Omron Sysmac Studio project Auto Connect Project (Sysmac Studio 1.61.0.64007, StandardProject)

# Controller new_Controller_0: NX102-9000 version 1.68
Units and slaves: 유니트 1 : NX-PF0730 (N1); 유니트 2 : NX-CIF105 (N2); 유니트 3 : NX-ID5342 (N3); 유니트 4 : NX-OD5121 (N4); 유니트 5 : NX-OD5121 (N5)
Task PrimaryTask (priority 4, period or condition 1000): Program0
Library MTCP_Server_NJNX 2.6. (contents left out)

TYPE sStepControl : STRUCT
    MoveStart : BOOL;
    TargetPulse : INT;  (* Unit : pulse *)
    SetDir : BOOL;  (* TRUE : CW, FALSE, CCW *)
END_STRUCT END_TYPE
TYPE sMotor : STRUCT
    Up : BOOL;
    Down : BOOL;
    Origin : BOOL;
    Move : INT;  (* Unit: 0.1 mm *)
    Check : BOOL;  (* Checking variable whether TRUE of FALSE *)
    Seq : INT;  (* Sequence Index *)
END_STRUCT END_TYPE
TYPE sModule : STRUCT
    Input : sModuleInput;
    Output : sModuleOutput;
END_STRUCT END_TYPE
TYPE sModuleInput : STRUCT
    Command : sModuleInputCommand;
END_STRUCT END_TYPE
TYPE sModuleOutput : STRUCT
    Status : sModuleOutputStatus;
END_STRUCT END_TYPE
TYPE sModuleInputCommand : STRUCT
    bCylinder1Down : BOOL;
    bCylinder1Up : BOOL;
END_STRUCT END_TYPE
TYPE sModuleOutputStatus : STRUCT
    bCylinder1Down : BOOL;
    bCylinder1Up : BOOL;
END_STRUCT END_TYPE

TYPE typeOPC\sProdTracker : STRUCT
    Input : typeOPC\sProdTrackerInput;
    Output : typeOPC\sProdTrackerOutput;
    Capture : typeOPC\sProdTrackerCapture;
    PTZ : typeOPC\sProdTrackerPTZ;
END_STRUCT END_TYPE
TYPE typeOPC\sProdTrackerInput : STRUCT
    nStart : INT;
    strData : STRING[256];
    nResult : INT;
END_STRUCT END_TYPE
TYPE typeOPC\sProdTrackerOutput : STRUCT
    nResponse : INT;
    dtUpdateTime : DATE_AND_TIME;
END_STRUCT END_TYPE
TYPE typeOPC\sProdTrackerCapture : STRUCT
    bStart : BOOL;
    strData : STRING[256];
END_STRUCT END_TYPE
TYPE typeOPC\sProdTrackerPTZ : STRUCT
    bStart : BOOL;
    nPreset : INT;
END_STRUCT END_TYPE

TYPE Data\sOT2 : STRUCT
    Pipette0 : INT;  (* 총 96개 pipette *)
    Pipette1 : INT;  (* 총 96개 pipette *)
    BigVial0 : Data\sBigVial;  (* 총 6개 바이알 *)
    BigVial1 : Data\sBigVial;  (* 총 6개 바이알 *)
    WellPlate : INT;  (* 총 96개 well *)
    HeatPlate : Data\sHeatPlate;  (* 총 12개 well *)
    OT2Job : STRING[256];  (* OT2 현황 *)
END_STRUCT END_TYPE
TYPE Data\sBigVial : STRUCT
    BVname : ARRAY[0..5] OF STRING[256];
    BVvolume : ARRAY[0..5] OF REAL;
END_STRUCT END_TYPE
TYPE Data\sHeatPlate : STRUCT
    HPname : ARRAY[0..11] OF STRING[256];
    HPvolume : ARRAY[0..11] OF REAL;
END_STRUCT END_TYPE
TYPE Data\sCell : STRUCT
    CSASstack : INT;  (* 양극, 스프링, 음극, 분리막 스태킹 구조물 (총 4개) *)
    CCSstack : INT;  (* 캔, 캡, 스페이서 스태킹 구조물 (총 4개) *)
    CScomp : INT;  (* 양극, 스프링 회전 구조물 (총 12개) *)
    AScomp : INT;  (* 음극, 분리막 회전 구조물 (총 12개) *)
    CCScomp : INT;  (* 캔, 캡, 스페이서 액츄에이터 구조물 (총 12개) *)
    Assembly : STRING[256];  (* 셀 조립대의 현황 (ex. can or sep or liquid) *)
    Crimper : BOOL;  (* 크림퍼 내 셀 존재 유무 *)
END_STRUCT END_TYPE
TYPE Data\sJig : STRUCT
    Cycler : Data\sCycler;
    EIS : Data\sEIS;
    Gantry : ARRAY[0..1] OF STRING[256];  (* 현재 직교로봇이 진행중인 작업 (ex. [EIS_Insert, 0]) *)
END_STRUCT END_TYPE
TYPE Data\sCycler : STRUCT
    name : ARRAY[0..47] OF STRING[256];  (* Cycling 셀 이름 *)
    status : ARRAY[0..47] OF STRING[256];  (* Cycler 현황 (empty, in, cycling, done) *)
END_STRUCT END_TYPE
TYPE Data\sEIS : STRUCT
    name : ARRAY[0..1] OF STRING[256];  (* EIS 셀 이름 *)
    status : ARRAY[0..1] OF STRING[256];  (* EIS 현황 (empty, in, cycling, done) *)
END_STRUCT END_TYPE

VAR_GLOBAL CONSTANT
    N1_Node_location_information : _sNXUNIT_ID := (NodeAdr := 65535, IPAdr := [5(16#FF)], UnitNo := 2, Path := [16#1, 16#0, 16#2, 16#0, 16#2, 59(16#0)], PathLength := 6);
END_VAR
VAR_GLOBAL
    Pulse0 : BOOL;  (* at IOBus://unit#5/Output Bit 16 bits/Output Bit 01 *)
    Direction0 : BOOL;  (* at IOBus://unit#5/Output Bit 16 bits/Output Bit 00 *)
    Pulse1 : BOOL;  (* at IOBus://unit#5/Output Bit 16 bits/Output Bit 03 *)
    Direction1 : BOOL;  (* at IOBus://unit#5/Output Bit 16 bits/Output Bit 02 *)
    Pulse2 : BOOL;  (* at IOBus://unit#5/Output Bit 16 bits/Output Bit 05 *)
    Direction2 : BOOL;  (* at IOBus://unit#5/Output Bit 16 bits/Output Bit 04 *)
    Pulse3 : BOOL;  (* at IOBus://unit#5/Output Bit 16 bits/Output Bit 07 *)
    Direction3 : BOOL;  (* at IOBus://unit#5/Output Bit 16 bits/Output Bit 06 *)
    Pulse4 : BOOL;  (* Front Z; at IOBus://unit#5/Output Bit 16 bits/Output Bit 09 *)
    Direction4 : BOOL;  (* Front Z; at IOBus://unit#5/Output Bit 16 bits/Output Bit 08 *)
    Pulse5 : BOOL;  (* Front X; at IOBus://unit#5/Output Bit 16 bits/Output Bit 11 *)
    Direction5 : BOOL;  (* Front X; at IOBus://unit#5/Output Bit 16 bits/Output Bit 10 *)
    Pulse6 : BOOL;  (* Back Z; at IOBus://unit#5/Output Bit 16 bits/Output Bit 13 *)
    Direction6 : BOOL;  (* Back Z; at IOBus://unit#5/Output Bit 16 bits/Output Bit 12 *)
    Pulse7 : BOOL;  (* Back X; at IOBus://unit#5/Output Bit 16 bits/Output Bit 15 *)
    Direction7 : BOOL;  (* Back X; at IOBus://unit#5/Output Bit 16 bits/Output Bit 14 *)
    Sensor0 : BOOL;  (* Rotary for Cathode&Spring; at IOBus://unit#3/Input Bit 16 bits/Input Bit 12 *)
    Sensor1 : BOOL;  (* Rotary for Anode&Separator; at IOBus://unit#3/Input Bit 16 bits/Input Bit 13 *)
    Sensor2 : BOOL;  (* Stacking for CSAS; at IOBus://unit#3/Input Bit 16 bits/Input Bit 14 *)
    Sensor3 : BOOL;  (* Stacking for Can&Cap&Spacer; at IOBus://unit#3/Input Bit 16 bits/Input Bit 15 *)
    Sensor4_L : BOOL;  (* Front Z; at IOBus://unit#3/Input Bit 16 bits/Input Bit 01 *)
    Sensor4_R : BOOL;  (* Front Z; at IOBus://unit#3/Input Bit 16 bits/Input Bit 02 *)
    Sensor5_L : BOOL;  (* Front X; at IOBus://unit#3/Input Bit 16 bits/Input Bit 04 *)
    Sensor5_R : BOOL;  (* Front X; at IOBus://unit#3/Input Bit 16 bits/Input Bit 05 *)
    Sensor6_L : BOOL;  (* Back Z; at IOBus://unit#3/Input Bit 16 bits/Input Bit 07 *)
    Sensor6_R : BOOL;  (* Back Z; at IOBus://unit#3/Input Bit 16 bits/Input Bit 08 *)
    Sensor7_L : BOOL;  (* Back X; at IOBus://unit#3/Input Bit 16 bits/Input Bit 10 *)
    Sensor7_R : BOOL;  (* Back X; at IOBus://unit#3/Input Bit 16 bits/Input Bit 11 *)
    ENA0 : BOOL;  (* at IOBus://unit#4/Output Bit 16 bits/Output Bit 01 *)
    ENA1 : BOOL;  (* at IOBus://unit#4/Output Bit 16 bits/Output Bit 03 *)
    ENA2 : BOOL;  (* at IOBus://unit#4/Output Bit 16 bits/Output Bit 05 *)
    ENA3 : BOOL;  (* at IOBus://unit#4/Output Bit 16 bits/Output Bit 07 *)
    ENA4 : BOOL;  (* at IOBus://unit#4/Output Bit 16 bits/Output Bit 09 *)
    ENA5 : BOOL;  (* at IOBus://unit#4/Output Bit 16 bits/Output Bit 11 *)
    ENA6 : BOOL;  (* at IOBus://unit#4/Output Bit 16 bits/Output Bit 13 *)
    ENA7 : BOOL;  (* at IOBus://unit#4/Output Bit 16 bits/Output Bit 15 *)
    RELAY0 : BOOL;  (* For STEP Motor; at IOBus://unit#4/Output Bit 16 bits/Output Bit 00 *)
    RELAY1 : BOOL;  (* For Crimper; at IOBus://unit#4/Output Bit 16 bits/Output Bit 02 *)
    Sensor4_O : BOOL;  (* Front Z *)
    Sensor5_O : BOOL;  (* Front X; at IOBus://unit#3/Input Bit 16 bits/Input Bit 03 *)
    Sensor6_O : BOOL;  (* Back Z; at IOBus://unit#3/Input Bit 16 bits/Input Bit 06 *)
    Sensor7_O : BOOL;  (* Back X; at IOBus://unit#3/Input Bit 16 bits/Input Bit 09 *)
    Robot_moving : BOOL;  (* True: Robot moving, False: Robot stop; at IOBus://unit#3/Input Bit 16 bits/Input Bit 00; published *)
    Motor0_Up : BOOL;  (* published *)
    Motor0_Down : BOOL;  (* published *)
    Motor0_Origin : BOOL;  (* published *)
    Motor0_Move : INT;  (* published *)
END_VAR
VAR_GLOBAL RETAIN
    Motor0_Check : BOOL;  (* published *)
END_VAR
VAR_GLOBAL
    Motor1_Up : BOOL;  (* published *)
    Motor1_Down : BOOL;  (* published *)
    Motor1_Origin : BOOL;  (* published *)
    Motor1_Move : INT;  (* published *)
    Motor1_Check : BOOL;  (* published *)
    Motor2_Up : BOOL;  (* published *)
    Motor2_Down : BOOL;  (* published *)
    Motor2_Origin : BOOL;  (* published *)
    Motor2_Move : INT;  (* published *)
    Motor2_Check : BOOL;  (* published *)
    Motor3_Up : BOOL;  (* published *)
    Motor3_Down : BOOL;  (* published *)
    Motor3_Origin : BOOL;  (* published *)
    Motor3_Move : INT;  (* published *)
    Motor3_Check : BOOL;  (* published *)
    Motor4_Up : BOOL;  (* published *)
    Motor4_Down : BOOL;  (* published *)
    Motor4_Origin : BOOL;  (* published *)
    Motor4_Move : INT;  (* 1 = 0.1 mm (ex. 25 = 2.5 mm); published *)
    Motor4_Check : BOOL;  (* published *)
    Motor5_Up : BOOL;  (* published *)
    Motor5_Down : BOOL;  (* published *)
    Motor5_Origin : BOOL;  (* published *)
    Motor5_Move : INT;  (* 1 = 0.1 mm (ex. 25 = 2.5 mm); published *)
    Motor5_Check : BOOL;  (* published *)
    Motor6_Up : BOOL;  (* published *)
    Motor6_Down : BOOL;  (* published *)
    Motor6_Origin : BOOL;  (* published *)
    Motor6_Move : INT;  (* 1 = 0.1 mm (ex. 25 = 2.5 mm); published *)
    Motor6_Check : BOOL;  (* published *)
    Motor7_Up : BOOL;  (* published *)
    Motor7_Down : BOOL;  (* published *)
    Motor7_Origin : BOOL;  (* published *)
    Motor7_Move : INT;  (* 1 = 0.1 mm (ex. 25 = 2.5 mm); published *)
    Motor7_Check : BOOL;  (* published *)
    Jigmove_csv : ARRAY[0..47,0..5] OF REAL;  (* for coincell Jig; published *)
    EISmove_csv : ARRAY[0..1,0..3] OF REAL;  (* for EIS Jig; published *)
    JigIndex : INT;  (* Jig: 0~47; published *)
    EISIndex : INT;  (* EIS: 0~1; published *)
    ActuIndex : INT;  (* published *)
    ActuMove : INT;  (* published *)
    Open_Serial : BOOL;  (* published *)
    PS2_Data : ARRAY[0..19] OF WORD;  (* Modbus TCP Write Data; published *)
    Open_MB : BOOL;  (* Modbus TCP Write; published *)
    Crimper_Done : BOOL;  (* published *)
    Crimper_On : BOOL;  (* published *)
    Jig_Readypos : BOOL;  (* published *)
    Jig_Insert : BOOL;  (* published *)
    Jig_Retrieve : BOOL;  (* published *)
    Robot_moving2 : BOOL;  (* 직접 지정 가능한 Robot moving Bool; published *)
    CCSactu_Check : BOOL;  (* 캔, 캡, 스페이서 액츄에이터 동작; published *)
    CCSactu_Index : INT;  (* 0: 원점, 1~12: 해당 위치만큼 올림; published *)
    CCSalign_Check : BOOL;  (* 캔, 캡, 스페이서 정렬 동작; published *)
    Assemalign_Check : BOOL;  (* 셀 조립대 정렬 동작; published *)
    JOBList : ARRAY[0..299] OF STRING[256];  (* 던져진 JOB 을 정리한 리스트; published *)
    JOB : ARRAY[0..1] OF STRING[256];  (* 지그에 던지는 JOB; published *)
    JOB_Done : BOOL;  (* True 면 지그에 던져진 다음 작업 수행; published *)
    Readypos_Done : BOOL;  (* 지그가 셀 받을 대기 상태; published *)
    Coincell_Job : ARRAY[0..47,0..9] OF BOOL;  (* 1열 셀 삽입(True: 셀 삽입됨), 2열: 1번 조건 완료, 3열: 2번 조건 완료...; published *)
    Coincell_EISJob : ARRAY[0..1,0..1] OF BOOL;  (* 1열 셀 삽입(True: 셀 삽입됨), 2열: 셀 평가 완료(True: 셀 평가 완료됨); published *)
    Coincell_Return : ARRAY[0..1] OF INT;  (* EIS 측정 후 돌아가야 할 포지션 위치; published *)
    ProdTracker : typeOPC\sProdTracker;  (* 카메라 (ProdTracker); published *)
    DataOT2 : Data\sOT2;  (* OT2 관련 데이터; published *)
    DataCell : Data\sCell;  (* 셀 조립 관련 데이터; published *)
    DataJig : Data\sJig;  (* 셀 지그 관련 데이터; published *)
END_VAR

PROGRAM Program0
VAR
    Open_Port : BOOL;
    Port_Open : BOOL;
    Port_Busy : BOOL;
    Port_Error : BOOL;
    Port_ErrorID : WORD;
    MB_Socket : _sSOCKET;
    do_nothing : BOOL;
    MBTCP_FN3 : ModbusTCPRead;
    Open_Socket : SktTCPConnect;
    FN3_Read_Cmd : _sMODBUS_READ;
    PS_Data : ARRAY[0..15] OF WORD;
    FN3_Busy : BOOL;
    FN3_Error : BOOL;
    FN3_ErrorID : WORD;
    FN3_Erridx : DWORD;
    Read_Size : UINT;
    do_nothing2 : BOOL;
    MBTCP_FN4 : ModbusTCPWrite;
    FN4_Write_Cmd : _sMODBUS_WRITE;
    FN4_Busy : BOOL;
    FN4_Error : BOOL;
    FN4_ErrorID : WORD;
    FN4_Erridx : DWORD;
    Open_RTU : BOOL;
    MBRTU_FN3 : NX_ModbusRtuWrite;
    MBRTU_FN1 : NX_ModbusRtuWrite;
    MBRTU_FN5 : NX_ModbusRtuWrite;
    FN5_Write_Cmd : _sSERIAL_MODBUSRTU_WRITE;
    PS5_Data : WORD;
    FN5_Port : _sDEVICE_PORT;
    FN5_Busy : BOOL;
    FN5_CmdAbort : BOOL;
    FN5_Error : BOOL;
    FN5_ErrorID : WORD;
    FN5_Erridx : DWORD;
    do_nothing3 : BOOL;
    RTUSlaveAdr : UINT := 11;
    bOutputStart : BOOL;
    bOutput : BOOL;
    nCount : INT;
    maxCount : INT;
    Open_Server : BOOL;
    TCPServer : MTCP_Server_NJNX;
    Server_Connected : BOOL;
    Reset_SdRcvCnt : BOOL := False;
    SdRcv_Cnt : UDINT;
    Port_Client : UINT;
    IP_Client : STRING[24];
    TCP_Status : _eCONNECTION_STATE;
    ErrorID : WORD;
    Error : BOOL;
    MotorStart : BOOL;
    TON_test : TON;
    TP_test : TP;
    FB_Motor1_Control : STEPmotor;
    Delay_TON0 : TON;
    o : BOOL;
    Motor1Control : sStepControl;
    FB_Motor0_Control : STEPmotor;
    Motor0Control : sStepControl;
    FB_Motor2_Control : STEPmotor;
    Motor2Control : sStepControl;
    Motor4Control : sStepControl;
    MotorRelay : BOOL;
    FB_Motor4_Control : STEPmotor;
    FB_Motor5_Control : STEPmotor;
    Motor5Control : sStepControl;
    FB_Motor6_Control : STEPmotor;
    Motor6Control : sStepControl;
    FB_Motor7_Control : STEPmotor;
    Motor7Control : sStepControl;
    Motor0 : sMotor;
    Motor1 : sMotor;
    Motor2 : sMotor;
    Motor3 : sMotor;
    Motor4 : sMotor;
    Motor5 : sMotor;
    Motor6 : sMotor;
    Motor7 : sMotor;
    FB_Motor3_Control : STEPmotor;
    Motor3Control : sStepControl;
    Open_MBRead : BOOL;
    bDebugBit : BOOL;
    Serial_FN6 : NX_SerialSend;
    do_nothing4 : BOOL;
    FN6_Port : _sDEVICE_PORT;
    Serial_Error : BOOL;
    Serial_Errid : WORD;
    Serial_Busy : BOOL;
    SendSize : UINT := 10;
    Jig_Origin : BOOL;
    Jig_Seq : INT;
    SendData : ARRAY[0..9] OF BYTE;
    JigOrigin_Seq : INT;
    chksum : BYTE;
    test : BOOL;
    Test_Seq : INT;
    JigReady_Seq : INT;
    Finish0 : BOOL;
    Finish1 : BOOL;
    Finish2 : BOOL;
    Finish3 : BOOL;
    Finish4 : BOOL;
    Finish5 : BOOL;
    Finish6 : BOOL;
    Finish7 : BOOL;
    JigRetrieve_Seq : INT;
    Crimper_Seq : INT;
    EIS_Seq : INT;
    EIS_Insert : BOOL;
    EISRetrieve_Seq : INT;
    EIS_Retrieve : BOOL;
    Delay_TON1 : TON;
    Delay_TON6 : TON;
    Delay_TON7 : TON;
    Delay_TON8 : TON;
    Delay_TON9 : TON;
    Delay_TON10 : TON;
    Delay_TON11 : TON;
    Delay_TON12 : TON;
    Delay_TON13 : TON;
    Delay_TON2 : TON;
    Delay_TON3 : TON;
    Delay_TON4 : TON;
    Delay_TON5 : TON;
    Delay_TON14 : TON;
    CCSactu_seq : INT;
    Delay_TON15 : TON;
    CCSalign_seq : INT;
    Delay_TON16 : TON;
    Assemalign_seq : INT;
    Delay_TON17 : TON;
    JOB_seq : INT;
    i : INT;
    JOBList_Clear : BOOL;
    JOBprocesstest : BOOL;
    JOBDone_Check : BOOL;
    SendData4 : BYTE := 05;
    SendData5 : BYTE := 243;
    SendData6 : BYTE := 134;
END_VAR
VAR_EXTERNAL CONSTANT
    N1_Node_location_information : _sNXUNIT_ID;
END_VAR
VAR_EXTERNAL
    Pulse0 : BOOL;
    Direction0 : BOOL;
    Pulse1 : BOOL;
    Direction1 : BOOL;
    ENA0 : BOOL;
    ENA1 : BOOL;
    ENA2 : BOOL;
    ENA3 : BOOL;
    ENA4 : BOOL;
    ENA5 : BOOL;
    ENA6 : BOOL;
    ENA7 : BOOL;
    RELAY0 : BOOL;
    Direction2 : BOOL;
    Direction3 : BOOL;
    Pulse2 : BOOL;
    Pulse3 : BOOL;
    Sensor0 : BOOL;
    Sensor1 : BOOL;
    Direction5 : BOOL;
    Pulse5 : BOOL;
    Sensor3 : BOOL;
    Sensor2 : BOOL;
    Direction4 : BOOL;
    Pulse4 : BOOL;
    Direction6 : BOOL;
    Pulse6 : BOOL;
    Direction7 : BOOL;
    Pulse7 : BOOL;
    Sensor4_L : BOOL;
    Sensor6_L : BOOL;
    Sensor4_R : BOOL;
    Sensor6_R : BOOL;
    Sensor5_L : BOOL;
    Sensor5_R : BOOL;
    Sensor7_L : BOOL;
    Sensor7_R : BOOL;
    Robot_moving : BOOL;
    Motor0_Up : BOOL;
    Motor0_Down : BOOL;
    Motor0_Origin : BOOL;
    Motor0_Move : INT;
    Motor0_Check : BOOL;
    Motor1_Up : BOOL;
    Motor1_Down : BOOL;
    Motor1_Origin : BOOL;
    Motor1_Move : INT;
    Motor1_Check : BOOL;
    Motor2_Up : BOOL;
    Motor2_Down : BOOL;
    Motor2_Origin : BOOL;
    Motor2_Move : INT;
    Motor2_Check : BOOL;
    Motor3_Up : BOOL;
    Motor3_Down : BOOL;
    Motor3_Origin : BOOL;
    Motor3_Move : INT;
    Motor3_Check : BOOL;
    Motor4_Up : BOOL;
    Motor4_Down : BOOL;
    Motor4_Origin : BOOL;
    Motor4_Move : INT;
    Motor4_Check : BOOL;
    Motor5_Up : BOOL;
    Motor5_Down : BOOL;
    Motor5_Origin : BOOL;
    Motor5_Move : INT;
    Motor5_Check : BOOL;
    Motor6_Up : BOOL;
    Motor6_Down : BOOL;
    Motor6_Origin : BOOL;
    Motor6_Move : INT;
    Motor6_Check : BOOL;
    Motor7_Up : BOOL;
    Motor7_Down : BOOL;
    Motor7_Origin : BOOL;
    Motor7_Move : INT;
    Motor7_Check : BOOL;
    Jigmove_csv : ARRAY[0..47,0..5] OF REAL;
    JigIndex : INT;
    ActuIndex : INT;
    ActuMove : INT;
    Open_Serial : BOOL;
    EISmove_csv : ARRAY[0..1,0..3] OF REAL;
    RELAY1 : BOOL;
    PS2_Data : ARRAY[0..19] OF WORD;
    Open_MB : BOOL;
    EISIndex : INT;
    Crimper_Done : BOOL;
    Crimper_On : BOOL;
    Jig_Readypos : BOOL;
    Jig_Insert : BOOL;
    Jig_Retrieve : BOOL;
    CCSactu_Check : BOOL;
    CCSactu_Index : INT;
    CCSalign_Check : BOOL;
    Assemalign_Check : BOOL;
    JOB : ARRAY[0..1] OF STRING[256];
    JOBList : ARRAY[0..299] OF STRING[256];
    JOB_Done : BOOL;
    Readypos_Done : BOOL;
    DataJig : Data\sJig;
END_VAR
VAR
    _e1 : R_TRIG;
    _e2 : R_TRIG;
    _e3 : R_TRIG;
    _p4 : BOOL;
END_VAR

(* Section Section0: ladder, written here as Structured Text *)

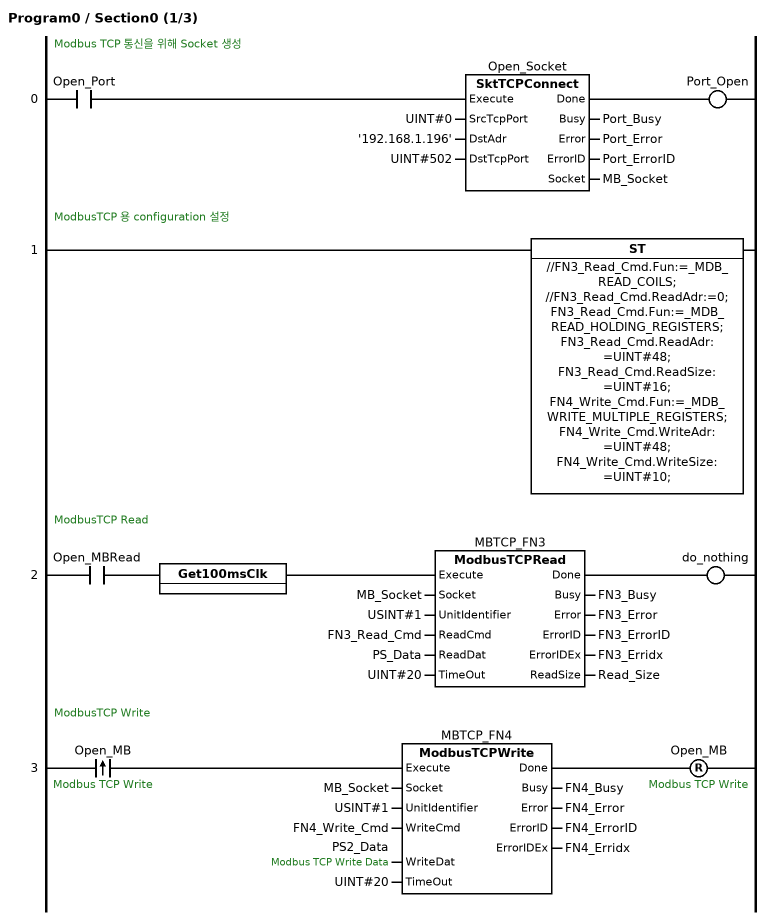
(* Rung 0: Modbus TCP 통신을 위해 Socket 생성 *)
Open_Socket(Execute := Open_Port, SrcTcpPort := UINT#0, DstAdr := '192.168.1.196', DstTcpPort := UINT#502, Busy => Port_Busy, Error => Port_Error, ErrorID => Port_ErrorID, Socket => MB_Socket);
Port_Open := Open_Socket.Done;
(* Rung 1: ModbusTCP 용 configuration 설정 *)
//FN3_Read_Cmd.Fun:=_MDB_READ_COILS;
//FN3_Read_Cmd.ReadAdr:=0;
FN3_Read_Cmd.Fun:=_MDB_READ_HOLDING_REGISTERS;
FN3_Read_Cmd.ReadAdr:=UINT#48;
FN3_Read_Cmd.ReadSize:=UINT#16;

FN4_Write_Cmd.Fun:=_MDB_WRITE_MULTIPLE_REGISTERS;
FN4_Write_Cmd.WriteAdr:=UINT#48;
FN4_Write_Cmd.WriteSize:=UINT#10;
(* Rung 2: ModbusTCP Read *)
MBTCP_FN3(Execute := Open_MBRead AND Get100msClk(), Socket := MB_Socket, UnitIdentifier := USINT#1, ReadCmd := FN3_Read_Cmd, ReadDat := PS_Data, TimeOut := UINT#20, Busy => FN3_Busy, Error => FN3_Error, ErrorID => FN3_ErrorID, ErrorIDEx => FN3_Erridx, ReadSize => Read_Size);
do_nothing := MBTCP_FN3.Done;
(* Rung 3: ModbusTCP Write *)
_e1(CLK := Open_MB);
MBTCP_FN4(Execute := _e1.Q, Socket := MB_Socket, UnitIdentifier := USINT#1, WriteCmd := FN4_Write_Cmd, WriteDat := PS2_Data, TimeOut := UINT#20, Busy => FN4_Busy, Error => FN4_Error, ErrorID => FN4_ErrorID, ErrorIDEx => FN4_Erridx);
IF MBTCP_FN4.Done THEN Open_MB := FALSE; END_IF;

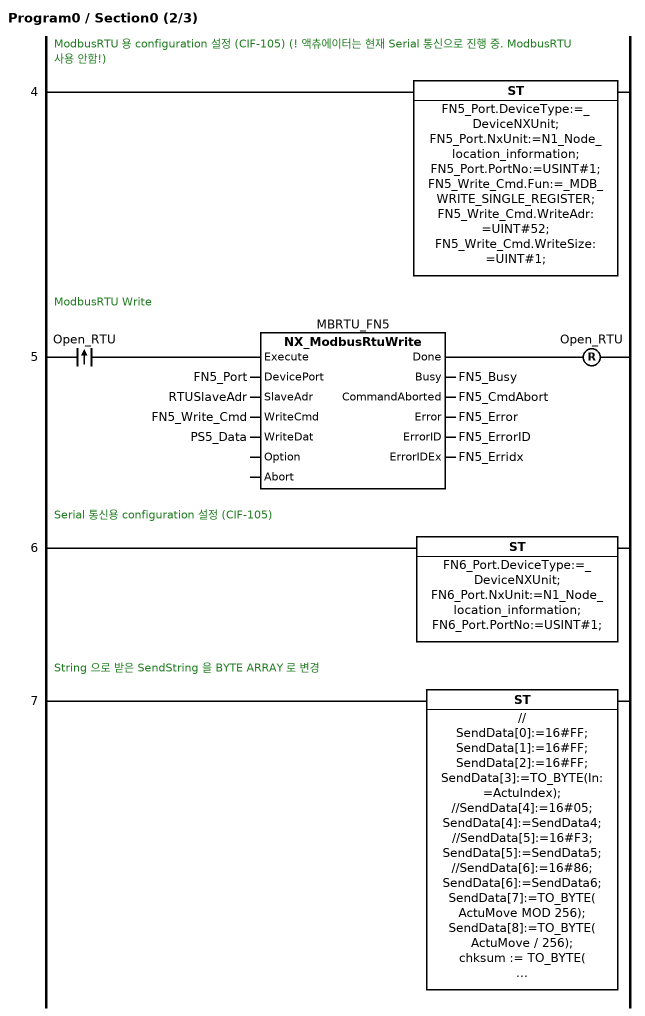
(* Rung 4: ModbusRTU 용 configuration 설정 (CIF-105) (! 액츄에이터는 현재 Serial 통신으로 진행 중. ModbusRTU 사용 안함!) *)
FN5_Port.DeviceType:=_DeviceNXUnit;
FN5_Port.NxUnit:=N1_Node_location_information;
FN5_Port.PortNo:=USINT#1;

FN5_Write_Cmd.Fun:=_MDB_WRITE_SINGLE_REGISTER;
FN5_Write_Cmd.WriteAdr:=UINT#52;
FN5_Write_Cmd.WriteSize:=UINT#1;
(* Rung 5: ModbusRTU Write *)
_e2(CLK := Open_RTU);
MBRTU_FN5(Execute := _e2.Q, DevicePort := FN5_Port, SlaveAdr := RTUSlaveAdr, WriteCmd := FN5_Write_Cmd, WriteDat := PS5_Data, Busy => FN5_Busy, CommandAborted => FN5_CmdAbort, Error => FN5_Error, ErrorID => FN5_ErrorID, ErrorIDEx => FN5_Erridx);
IF MBRTU_FN5.Done THEN Open_RTU := FALSE; END_IF;
(* Rung 6: Serial 통신용 configuration 설정 (CIF-105) *)
FN6_Port.DeviceType:=_DeviceNXUnit;
FN6_Port.NxUnit:=N1_Node_location_information;
FN6_Port.PortNo:=USINT#1;
(* Rung 7: String 으로 받은 SendString 을 BYTE ARRAY 로 변경 *)
// 
SendData[0]:=16#FF;
SendData[1]:=16#FF;
SendData[2]:=16#FF;

SendData[3]:=TO_BYTE(In:=ActuIndex);
//SendData[4]:=16#05;
SendData[4]:=SendData4;
//SendData[5]:=16#F3;
SendData[5]:=SendData5;

//SendData[6]:=16#86;
SendData[6]:=SendData6;

SendData[7]:=TO_BYTE(ActuMove MOD 256);
SendData[8]:=TO_BYTE(ActuMove / 256);
chksum := TO_BYTE(
			  255 -
			  (TO_INT(SendData[3])
			  + TO_INT(SendData[4])
			  + TO_INT(SendData[5])
			  + TO_INT(SendData[6])
			  + TO_INT(SendData[7])
			  + TO_INT(SendData[8])));

SendData[9] := chksum;

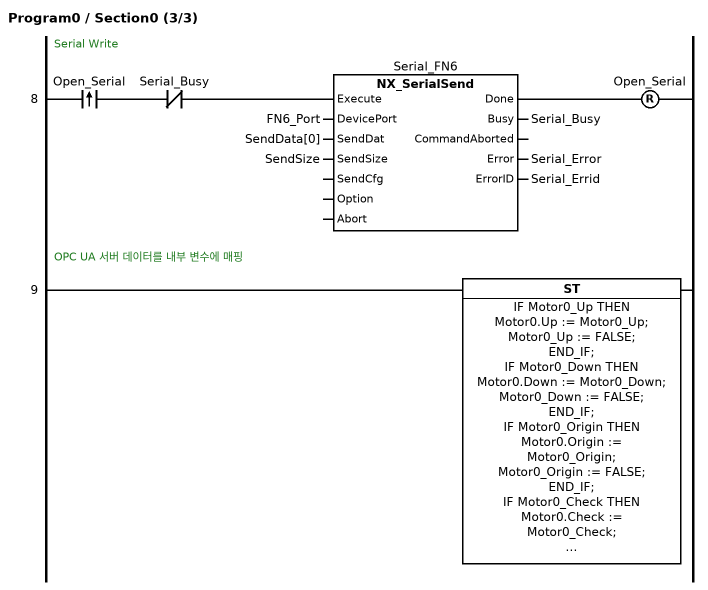
(* Rung 8: Serial Write *)
_e3(CLK := Open_Serial);
_p4 := _e3.Q AND NOT Serial_Busy;
Serial_FN6(Execute := _p4, DevicePort := FN6_Port, SendDat := SendData[0], SendSize := SendSize, Busy => Serial_Busy, Error => Serial_Error, ErrorID => Serial_Errid);
IF Serial_FN6.Done THEN Open_Serial := FALSE; END_IF;
(* Rung 9: OPC UA 서버 데이터를 내부 변수에 매핑 *)
IF Motor0_Up THEN
    Motor0.Up := Motor0_Up;
    Motor0_Up := FALSE;
END_IF;
IF Motor0_Down THEN
    Motor0.Down := Motor0_Down;
    Motor0_Down := FALSE;
END_IF;
IF Motor0_Origin THEN
    Motor0.Origin := Motor0_Origin;
    Motor0_Origin := FALSE;
END_IF;
IF Motor0_Check THEN
    Motor0.Check := Motor0_Check;
    Motor0_Check := FALSE;
END_IF;

IF Motor1_Up THEN
    Motor1.Up := Motor1_Up;
    Motor1_Up := FALSE;
END_IF;
IF Motor1_Down THEN
    Motor1.Down := Motor1_Down;
    Motor1_Down := FALSE;
END_IF;
IF Motor1_Origin THEN
    Motor1.Origin := Motor1_Origin;
    Motor1_Origin := FALSE;
END_IF;
IF Motor1_Check THEN
    Motor1.Check := Motor1_Check;
    Motor1_Check := FALSE;
END_IF;

IF Motor2_Up THEN
    Motor2.Up := Motor2_Up;
    Motor2_Up := FALSE;
END_IF;
IF Motor2_Down THEN
    Motor2.Down := Motor2_Down;
    Motor2_Down := FALSE;
END_IF;
IF Motor2_Origin THEN
    Motor2.Origin := Motor2_Origin;
    Motor2_Origin := FALSE;
END_IF;
IF Motor2_Check THEN
    Motor2.Check := Motor2_Check;
    Motor2_Check := FALSE;
END_IF;

IF Motor3_Up THEN
    Motor3.Up := Motor3_Up;
    Motor3_Up := FALSE;
END_IF;
IF Motor3_Down THEN
    Motor3.Down := Motor3_Down;
    Motor3_Down := FALSE;
END_IF;
IF Motor3_Origin THEN
    Motor3.Origin := Motor3_Origin;
    Motor3_Origin := FALSE;
END_IF;
IF Motor3_Check THEN
    Motor3.Check := Motor3_Check;
    Motor3_Check := FALSE;
END_IF;

IF Motor4_Up THEN
    Motor4.Up := Motor4_Up;
    Motor4_Up := FALSE;
END_IF;
IF Motor4_Down THEN
    Motor4.Down := Motor4_Down;
    Motor4_Down := FALSE;
END_IF;
IF Motor4_Origin THEN
    Motor4.Origin := Motor4_Origin;
    Motor4_Origin := FALSE;
END_IF;
IF Motor4_Check THEN
    Motor4.Check := Motor4_Check;
    Motor4_Check := FALSE;
END_IF;

IF Motor5_Up THEN
    Motor5.Up := Motor5_Up;
    Motor5_Up := FALSE;
END_IF;
IF Motor5_Down THEN
    Motor5.Down := Motor5_Down;
    Motor5_Down := FALSE;
END_IF;
IF Motor5_Origin THEN
    Motor5.Origin := Motor5_Origin;
    Motor5_Origin := FALSE;
END_IF;
IF Motor5_Check THEN
    Motor5.Check := Motor5_Check;
    Motor5_Check := FALSE;
END_IF;

IF Motor6_Up THEN
    Motor6.Up := Motor6_Up;
    Motor6_Up := FALSE;
END_IF;
IF Motor6_Down THEN
    Motor6.Down := Motor6_Down;
    Motor6_Down := FALSE;
END_IF;
IF Motor6_Origin THEN
    Motor6.Origin := Motor6_Origin;
    Motor6_Origin := FALSE;
END_IF;
IF Motor6_Check THEN
    Motor6.Check := Motor6_Check;
    Motor6_Check := FALSE;
END_IF;

IF Motor7_Up THEN
    Motor7.Up := Motor7_Up;
    Motor7_Up := FALSE;
END_IF;
IF Motor7_Down THEN
    Motor7.Down := Motor7_Down;
    Motor7_Down := FALSE;
END_IF;
IF Motor7_Origin THEN
    Motor7.Origin := Motor7_Origin;
    Motor7_Origin := FALSE;
END_IF;
IF Motor7_Check THEN
    Motor7.Check := Motor7_Check;
    Motor7_Check := FALSE;
END_IF;

Motor0.Move := Motor0_Move;
Motor1.Move := Motor1_Move;
Motor2.Move := Motor2_Move;
Motor3.Move := Motor3_Move;
Motor4.Move := Motor4_Move;
Motor5.Move := Motor5_Move;
Motor6.Move := Motor6_Move;
Motor7.Move := Motor7_Move;

(* Section Section1: ladder, written here as Structured Text *)

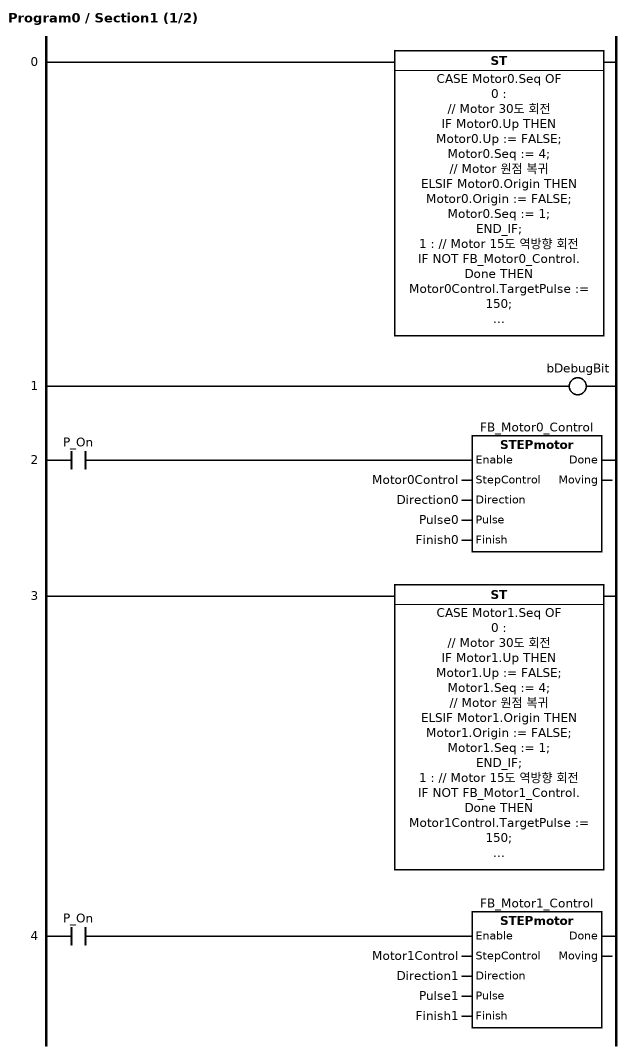
(* Rung 0 *)
CASE Motor0.Seq OF
	
	0 : 
		// Motor 30도 회전
		IF Motor0.Up THEN
			Motor0.Up := FALSE;
			Motor0.Seq := 4;
		// Motor 원점 복귀
		ELSIF Motor0.Origin THEN
			Motor0.Origin := FALSE;
			Motor0.Seq := 1;
		END_IF;
		
	1 : // Motor 15도 역방향 회전
		IF NOT FB_Motor0_Control.Done THEN
			Motor0Control.TargetPulse := 150;
			Motor0Control.SetDir	:= TRUE;
			Motor0Control.MoveStart := TRUE;
		END_IF;
		
		IF FB_Motor0_Control.Done THEN
			Motor0Control.MoveStart := FALSE;
			Motor0.Seq := 2;
		END_IF;
		
	2: // 0.5s delay
		Delay_TON0.In := TRUE;
		Delay_TON0.PT := T#0.5s;
		Delay_TON0();
		
		IF Delay_TON0.Q THEN
			Delay_TON0.In := FALSE;
			Delay_TON0();
			Motor0.Seq := 3;
		END_IF;
			
	3 : // 원점까지 Motor 정방향 회전
		IF NOT FB_Motor0_Control.Done AND NOT Sensor0 THEN
			Motor0Control.TargetPulse := 3600;
			Motor0Control.SetDir	:= FALSE;
			Motor0Control.MoveStart := TRUE;
		ELSE
			Motor0Control.MoveStart := FALSE;
			Motor0.Seq := 0;
		END_IF;
		
	4: // Motor 정방향 30도 회전 
		IF NOT FB_Motor0_Control.Done THEN
			Motor0Control.TargetPulse := 300;
			Motor0Control.SetDir := FALSE;
			Motor0Control.MoveStart:=TRUE;
		END_IF;
		
		IF FB_Motor0_Control.Done THEN
			Motor0Control.MoveStart := FALSE;
			Motor0.Seq := 0;
		END_IF;
	
END_CASE;
(* Rung 1 *)
bDebugBit := TRUE;
(* Rung 2 *)
FB_Motor0_Control(Enable := P_On, StepControl := Motor0Control, Direction := Direction0, Pulse := Pulse0, Finish := Finish0);
(* Rung 3 *)
CASE Motor1.Seq OF
	
	0 : 
		// Motor 30도 회전
		IF Motor1.Up THEN
			Motor1.Up := FALSE;
			Motor1.Seq := 4;
		// Motor 원점 복귀
		ELSIF Motor1.Origin THEN
			Motor1.Origin := FALSE;
			Motor1.Seq := 1;
		END_IF;
		
	1 : // Motor 15도 역방향 회전
		IF NOT FB_Motor1_Control.Done THEN
			Motor1Control.TargetPulse := 150;
			Motor1Control.SetDir	:= FALSE;
			Motor1Control.MoveStart := TRUE;
		END_IF;
		
		IF FB_Motor1_Control.Done THEN
			Motor1Control.MoveStart := FALSE;
			Motor1.Seq := 2;
		END_IF;
		
	2: // 0.5s delay
		Delay_TON1.In := TRUE;
		Delay_TON1.PT := T#0.5s;
		Delay_TON1();
		
		IF Delay_TON1.Q THEN
			Delay_TON1.In := FALSE;
			Delay_TON1();
			Motor1.Seq := 3;
		END_IF;
			
	3 : // 원점까지 Motor 정방향 회전
		IF NOT FB_Motor1_Control.Done AND NOT Sensor1 THEN
			Motor1Control.TargetPulse := 3600;
			Motor1Control.SetDir	:= TRUE;
			Motor1Control.MoveStart := TRUE;
		ELSE
			Motor1Control.MoveStart := FALSE;
			Motor1.Seq := 0;
		END_IF;
		
	4: // Motor 정방향 30도 회전 
		IF NOT FB_Motor1_Control.Done THEN
			Motor1Control.TargetPulse := 300;
			Motor1Control.SetDir := TRUE;
			Motor1Control.MoveStart:=TRUE;
		END_IF;
		
		IF FB_Motor1_Control.Done THEN
			Motor1Control.MoveStart := FALSE;
			Motor1.Seq := 0;
		END_IF;
	
END_CASE;
(* Rung 4 *)
FB_Motor1_Control(Enable := P_On, StepControl := Motor1Control, Direction := Direction1, Pulse := Pulse1, Finish := Finish1);

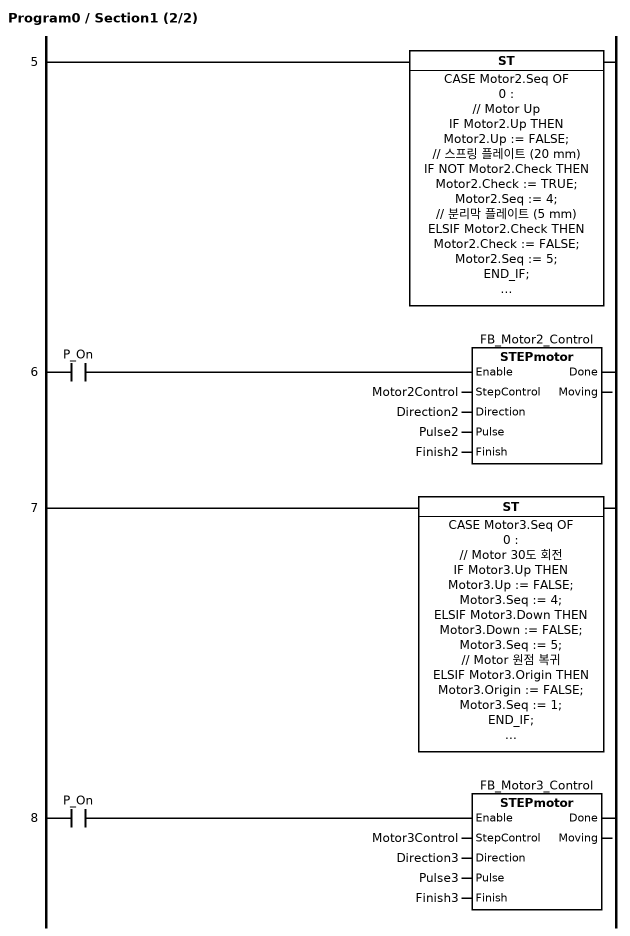
(* Rung 5 *)
CASE Motor2.Seq OF
	
	0 : 
		// Motor Up
		IF Motor2.Up THEN
			Motor2.Up := FALSE;
			// 스프링 플레이트 (20 mm)
			IF NOT Motor2.Check THEN
				Motor2.Check := TRUE;
				Motor2.Seq := 4;
			// 분리막 플레이트 (5 mm)
			ELSIF Motor2.Check THEN
				Motor2.Check := FALSE;
				Motor2.Seq := 5;
			END_IF;
		ELSIF Motor2.Down THEN
			Motor2.Down := FALSE;
			IF Motor2.Check THEN
				Motor2.Check := FALSE;
				Motor2.Seq := 6;
			ELSIF NOT Motor2.Check THEN
				Motor2.Check := TRUE;
				Motor2.Seq := 7;
			END_IF;
		// Motor 원점 복귀
		ELSIF Motor2.Origin THEN
			Motor2.Origin := FALSE;
			Motor2.Check := FALSE;
			Motor2.Seq := 1;
		END_IF;
		
	1 : // Motor 15도 역방향 회전
		IF NOT FB_Motor2_Control.Done THEN
			Motor2Control.TargetPulse := 50;
			Motor2Control.SetDir	:= FALSE;
			Motor2Control.MoveStart := TRUE;
		END_IF;
		
		IF FB_Motor2_Control.Done THEN
			Motor2Control.MoveStart := FALSE;
			Motor2.Seq := 2;
		END_IF;
		
	2: // 0.5s delay
		Delay_TON2.In := TRUE;
		Delay_TON2.PT := T#0.5s;
		Delay_TON2();
		
		IF Delay_TON2.Q THEN
			Delay_TON2.In := FALSE;
			Delay_TON2();
			Motor2.Seq := 3;
		END_IF;
			
	3 : // 원점까지 Motor 정방향 회전
		IF NOT FB_Motor2_Control.Done AND NOT Sensor2 THEN
			Motor2Control.TargetPulse := 10050;
			Motor2Control.SetDir	:= TRUE;
			Motor2Control.MoveStart := TRUE;
		ELSE
			Motor2Control.MoveStart := FALSE;
			Motor2.Seq := 0;
		END_IF;
		
	4: // Motor 
		IF NOT FB_Motor2_Control.Done THEN
			Motor2Control.TargetPulse := 2000;
			Motor2Control.SetDir := FALSE;
			Motor2Control.MoveStart:=TRUE;
		END_IF;
		
		IF FB_Motor2_Control.Done THEN
			Motor2Control.MoveStart := FALSE;
			Motor2.Seq := 0;
		END_IF;
		
	5:
		IF NOT FB_Motor2_Control.Done THEN
			Motor2Control.TargetPulse := 500;
			Motor2Control.SetDir := FALSE;
			Motor2Control.MoveStart:=TRUE;
		END_IF;
		
		IF FB_Motor2_Control.Done THEN
			Motor2Control.MoveStart := FALSE;
			Motor2.Seq := 0;
		END_IF;
		
	6:
		IF NOT FB_Motor2_Control.Done THEN
			Motor2Control.TargetPulse := 2000;
			Motor2Control.SetDir := TRUE;
			Motor2Control.MoveStart:=TRUE;
		END_IF;
		
		IF FB_Motor2_Control.Done THEN
			Motor2Control.MoveStart := FALSE;
			Motor2.Seq := 0;
		END_IF;

	7:
		IF NOT FB_Motor2_Control.Done THEN
			Motor2Control.TargetPulse := 500;
			Motor2Control.SetDir := TRUE;
			Motor2Control.MoveStart:=TRUE;
		END_IF;
	
		IF FB_Motor2_Control.Done THEN
			Motor2Control.MoveStart := FALSE;
			Motor2.Seq := 0;
		END_IF;
		
	
END_CASE;
(* Rung 6 *)
FB_Motor2_Control(Enable := P_On, StepControl := Motor2Control, Direction := Direction2, Pulse := Pulse2, Finish := Finish2);
(* Rung 7 *)
CASE Motor3.Seq OF
	
	0 : 
		// Motor 30도 회전
		IF Motor3.Up THEN
			Motor3.Up := FALSE;
			Motor3.Seq := 4;
		ELSIF Motor3.Down THEN
			Motor3.Down := FALSE;
			Motor3.Seq := 5;
		// Motor 원점 복귀
		ELSIF Motor3.Origin THEN
			Motor3.Origin := FALSE;
			Motor3.Seq := 1;
		END_IF;
		
	1 : // Motor 15도 역방향 회전
		IF NOT FB_Motor3_Control.Done THEN
			Motor3Control.TargetPulse := 50;
			Motor3Control.SetDir	:= FALSE;
			Motor3Control.MoveStart := TRUE;
		END_IF;
		
		IF FB_Motor3_Control.Done THEN
			Motor3Control.MoveStart := FALSE;
			Motor3.Seq := 2;
		END_IF;
		
	2: // 0.5s delay
		Delay_TON3.In := TRUE;
		Delay_TON3.PT := T#0.5s;
		Delay_TON3();
		
		IF Delay_TON3.Q THEN
			Delay_TON3.In := FALSE;
			Delay_TON3();
			Motor3.Seq := 3;
		END_IF;
			
	3 : // 원점까지 Motor 정방향 회전
		IF NOT FB_Motor3_Control.Done AND NOT Sensor3 THEN
			Motor3Control.TargetPulse := 16050;
			Motor3Control.SetDir	:= TRUE;
			Motor3Control.MoveStart := TRUE;
		ELSE
			Motor3Control.MoveStart := FALSE;
			Motor3.Seq := 0;
		END_IF;
		
	4: // Motor 
		IF NOT FB_Motor3_Control.Done THEN
			Motor3Control.TargetPulse := 4000;
			Motor3Control.SetDir := FALSE;
			Motor3Control.MoveStart:=TRUE;
		END_IF;
		
		IF FB_Motor3_Control.Done THEN
			Motor3Control.MoveStart := FALSE;
			Motor3.Seq := 0;
		END_IF;
		
	5: // Motor 
		IF NOT FB_Motor3_Control.Done THEN
			Motor3Control.TargetPulse := 4000;
			Motor3Control.SetDir := TRUE;
			Motor3Control.MoveStart:=TRUE;
		END_IF;
		
		IF FB_Motor3_Control.Done THEN
			Motor3Control.MoveStart := FALSE;
			Motor3.Seq := 0;
		END_IF;
	
END_CASE;
(* Rung 8 *)
FB_Motor3_Control(Enable := P_On, StepControl := Motor3Control, Direction := Direction3, Pulse := Pulse3, Finish := Finish3);

(* Section Section2: ladder, written here as Structured Text *)

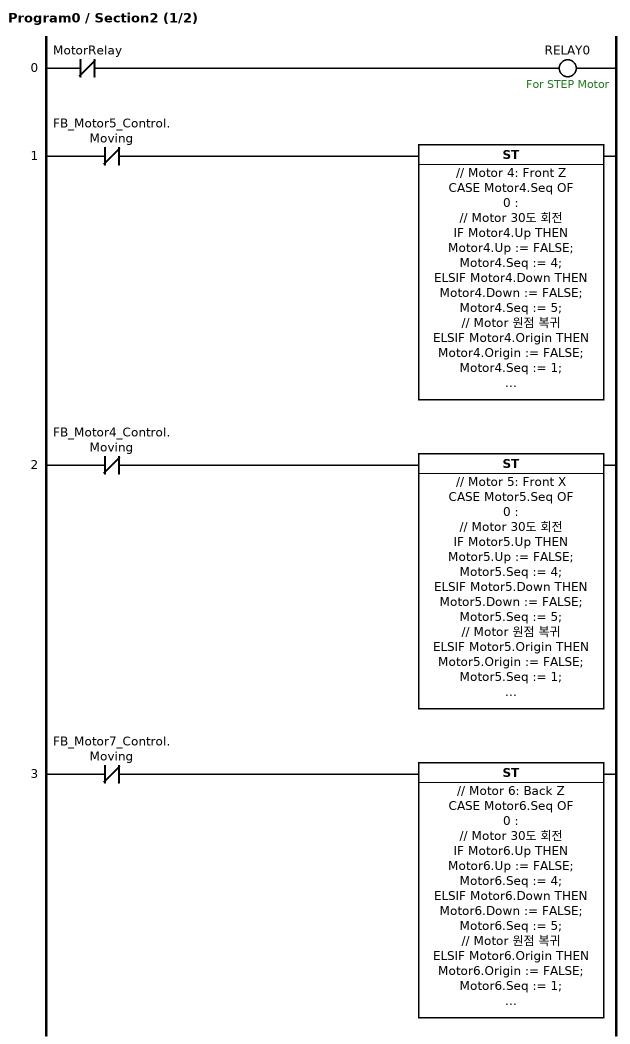
(* Rung 0 *)
RELAY0 := NOT MotorRelay;
(* Rung 1 *)
IF NOT FB_Motor5_Control.Moving THEN
    // Motor 4: Front Z
    	
    CASE Motor4.Seq OF
    	
    	0 : 
    		// Motor 30도 회전
    		IF Motor4.Up THEN
    			Motor4.Up := FALSE;
    			Motor4.Seq := 4;
    		ELSIF Motor4.Down THEN
    			Motor4.Down := FALSE;
    			Motor4.Seq := 5;
    		// Motor 원점 복귀
    		ELSIF Motor4.Origin THEN
    			Motor4.Origin := FALSE;
    			Motor4.Seq := 1;
    		// Motor.Check 가 TRUE 면 Motor.Move 에 설정된 거리만큼 이동
    		ELSIF Motor4.Check THEN
    			Motor4.Check := FALSE;
    			Motor4.Seq := 6;
    		
    		END_IF;
    		
    		
    	1 : // Motor 15도 역방향 회전
    		IF NOT FB_Motor4_Control.Done THEN
    			Motor4Control.TargetPulse := 50;
    			Motor4Control.SetDir	:= TRUE;
    			Motor4Control.MoveStart := TRUE;
    			Finish4:=FALSE;
    		END_IF;
    		
    		IF FB_Motor4_Control.Done THEN
    			Motor4Control.MoveStart := FALSE;
    			Motor4.Seq := 2;
    		END_IF;
    		
    	2: // 0.5s delay
    		Delay_TON4.In := TRUE;
    		Delay_TON4.PT := T#0.5s;
    		Delay_TON4();
    		
    		IF Delay_TON4.Q THEN
    			Delay_TON4.In := FALSE;
    			Delay_TON4();
    			Motor4.Seq := 3;
    		END_IF;
    			
    	3 : // 원점까지 Motor 정방향 회전
    		IF NOT FB_Motor4_Control.Done AND NOT Sensor4_L THEN
    			Motor4Control.TargetPulse := 20000;
    			Motor4Control.SetDir	:= FALSE;
    			Motor4Control.MoveStart := TRUE;
    		ELSE
    			Motor4Control.MoveStart := FALSE;
    			Motor4.Seq := 7;
    		END_IF;
    		
    	4: // Motor 
    		IF NOT FB_Motor4_Control.Done AND NOT Sensor4_L THEN
    			Motor4Control.TargetPulse := 1375;
    			Motor4Control.SetDir := FALSE;
    			Motor4Control.MoveStart:=TRUE;
    		END_IF;
    		
    		IF FB_Motor4_Control.Done THEN
    			Motor4Control.MoveStart := FALSE;
    			Motor4.Seq := 0;
    		END_IF;
    		
    	5: // Motor 
    		IF NOT FB_Motor4_Control.Done AND NOT Sensor4_R THEN
    			Motor4Control.TargetPulse := 1375;
    			Motor4Control.SetDir := TRUE;
    			Motor4Control.MoveStart:=TRUE;
    		END_IF;
    		
    		IF FB_Motor4_Control.Done THEN
    			Motor4Control.MoveStart := FALSE;
    			Motor4.Seq := 0;
    		END_IF;
    	
    	6: // 지정 거리 이동
    		IF NOT FB_Motor4_Control.Done AND NOT Sensor4_L AND NOT Sensor4_R THEN
    			IF Motor4.Move >= 0 THEN
    				Motor4Control.SetDir := TRUE;
    			ELSIF Motor4.Move < 0 THEN
    				Motor4Control.SetDir := FALSE;
    			END_IF;
    			
    			Motor4Control.TargetPulse := ABS(Motor4.Move)*200/80;
    			Motor4Control.MoveStart := TRUE;
    			Finish4:=FALSE;
    		END_IF;
    		
    		IF FB_Motor4_Control.Done THEN
    			Motor4Control.MoveStart := FALSE;
    			Finish4:=TRUE;
    			Motor4.Seq := 0;
    		END_IF;
    	
    	7: // LSL 도달 시 복귀
    		IF NOT FB_Motor4_Control.Done AND Sensor4_L THEN
    			Motor4Control.TargetPulse := 350;
    			Motor4Control.SetDir := TRUE;
    			Motor4Control.MoveStart := TRUE;
    		END_IF;
    		
    		IF FB_Motor4_Control.Done THEN
    			Motor4Control.MoveStart := FALSE;
    			Finish4:=TRUE;
    			Motor4.Seq := 0;
    		END_IF;
    		
    	8: // RSL 도달 시 복귀
    		IF NOT FB_Motor4_Control.Done AND Sensor4_R THEN
    			Motor4Control.TargetPulse := 180;
    			Motor4Control.SetDir := FALSE;
    			Motor4Control.MoveStart := TRUE;
    		END_IF;
    		
    		IF FB_Motor4_Control.Done THEN
    			Motor4Control.MoveStart := FALSE;
    			Motor4.Seq := 0;
    		END_IF;
    END_CASE;
END_IF;
(* Rung 2 *)
IF NOT FB_Motor4_Control.Moving THEN
    // Motor 5: Front X
    
    CASE Motor5.Seq OF
    	
    	0 : 
    		// Motor 30도 회전
    		IF Motor5.Up THEN
    			Motor5.Up := FALSE;
    			Motor5.Seq := 4;
    		ELSIF Motor5.Down THEN
    			Motor5.Down := FALSE;
    			Motor5.Seq := 5;
    		// Motor 원점 복귀
    		ELSIF Motor5.Origin THEN
    			Motor5.Origin := FALSE;
    			Motor5.Seq := 1;
    		// Motor.Check 가 TRUE 면 Motor.Move 에 설정된 거리만큼 이동
    		ELSIF Motor5.Check THEN
    			Motor5.Check := FALSE;
    			Motor5.Seq := 6;
    		
    		END_IF;
    		
    		
    	1 : // Motor 15도 역방향 회전
    		IF NOT FB_Motor5_Control.Done THEN
    			Motor5Control.TargetPulse := 50;
    			Motor5Control.SetDir	:= FALSE;
    			Motor5Control.MoveStart := TRUE;
    			Finish5:=FALSE;
    		END_IF;
    		
    		IF FB_Motor5_Control.Done THEN
    			Motor5Control.MoveStart := FALSE;
    			Motor5.Seq := 2;
    		END_IF;
    		
    	2: // 0.5s delay
    		Delay_TON5.In := TRUE;
    		Delay_TON5.PT := T#0.5s;
    		Delay_TON5();
    		
    		IF Delay_TON5.Q THEN
    			Delay_TON5.In := FALSE;
    			Delay_TON5();
    			Motor5.Seq := 3;
    		END_IF;
    			
    	3 : // 원점까지 Motor 정방향 회전
    		IF NOT FB_Motor5_Control.Done AND NOT Sensor5_L THEN
    			Motor5Control.TargetPulse := 20000;
    			Motor5Control.SetDir	:= TRUE;
    			Motor5Control.MoveStart := TRUE;
    		ELSE
    			Motor5Control.MoveStart := FALSE;
    			Motor5.Seq := 7;
    		END_IF;
    		
    	4: // Motor 
    		IF NOT FB_Motor5_Control.Done AND NOT Sensor5_L THEN
    			Motor5Control.TargetPulse := 900;
    			Motor5Control.SetDir := FALSE;
    			Motor5Control.MoveStart:=TRUE;
    		END_IF;
    		
    		IF FB_Motor5_Control.Done THEN
    			Motor5Control.MoveStart := FALSE;
    			Motor5.Seq := 0;
    		END_IF;
    		
    	5: // Motor 
    		IF NOT FB_Motor5_Control.Done AND NOT Sensor5_R THEN
    			Motor5Control.TargetPulse := 900;
    			Motor5Control.SetDir := TRUE;
    			Motor5Control.MoveStart:=TRUE;
    		END_IF;
    		
    		IF FB_Motor5_Control.Done THEN
    			Motor5Control.MoveStart := FALSE;
    			Motor5.Seq := 0;
    		END_IF;
    	
    	6: // 지정 거리 이동
    		IF NOT FB_Motor5_Control.Done AND NOT Sensor5_L AND NOT Sensor5_R THEN
    			IF Motor5.Move >= 0 THEN
    				Motor5Control.SetDir := FALSE;
    			ELSIF Motor5.Move < 0 THEN
    				Motor5Control.SetDir := TRUE;
    			END_IF;
    			
    			Motor5Control.TargetPulse := ABS(Motor5.Move)*200/100;
    			Motor5Control.MoveStart := TRUE;
    			Finish5:=FALSE;
    		END_IF;
    		
    		IF FB_Motor5_Control.Done THEN
    			Motor5Control.MoveStart := FALSE;
    			Finish5:=TRUE;
    			Motor5.Seq := 0;
    		END_IF;
    	
    	7: // LSL 도달 시 복귀
    		IF NOT FB_Motor5_Control.Done AND Sensor5_L THEN
    			Motor5Control.TargetPulse := 140;
    			Motor5Control.SetDir := FALSE;
    			Motor5Control.MoveStart := TRUE;
    		END_IF;
    		
    		IF FB_Motor5_Control.Done THEN
    			Motor5Control.MoveStart := FALSE;
    			Finish5:=TRUE;
    			Motor5.Seq := 0;
    		END_IF;
    		
    		8: // LSL 도달 시 복귀
    		IF NOT FB_Motor5_Control.Done AND Sensor5_R THEN
    			Motor5Control.TargetPulse := 180;
    			Motor5Control.SetDir := TRUE;
    			Motor5Control.MoveStart := TRUE;
    		END_IF;
    		
    		IF FB_Motor5_Control.Done THEN
    			Motor5Control.MoveStart := FALSE;
    			Motor5.Seq := 0;
    		END_IF;
    END_CASE;
END_IF;
(* Rung 3 *)
IF NOT FB_Motor7_Control.Moving THEN
    // Motor 6: Back Z
    
    CASE Motor6.Seq OF
    	
    	0 : 
    		// Motor 30도 회전
    		IF Motor6.Up THEN
    			Motor6.Up := FALSE;
    			Motor6.Seq := 4;
    		ELSIF Motor6.Down THEN
    			Motor6.Down := FALSE;
    			Motor6.Seq := 5;
    		// Motor 원점 복귀
    		ELSIF Motor6.Origin THEN
    			Motor6.Origin := FALSE;
    			Motor6.Seq := 1;
    		// Motor.Check 가 TRUE 면 Motor.Move 에 설정된 거리만큼 이동
    		ELSIF Motor6.Check THEN
    			Motor6.Check := FALSE;
    			Motor6.Seq := 6;
    		
    		END_IF;
    		
    		
    	1 : // Motor 15도 역방향 회전
    		IF NOT FB_Motor6_Control.Done THEN
    			Motor6Control.TargetPulse := 50;
    			Motor6Control.SetDir	:= TRUE;
    			Motor6Control.MoveStart := TRUE;
    			Finish6:=FALSE;
    		END_IF;
    		
    		IF FB_Motor6_Control.Done THEN
    			Motor6Control.MoveStart := FALSE;
    			Motor6.Seq := 2;
    		END_IF;
    		
    	2: // 0.5s delay
    		Delay_TON6.In := TRUE;
    		Delay_TON6.PT := T#0.5s;
    		Delay_TON6();
    		
    		IF Delay_TON6.Q THEN
    			Delay_TON6.In := FALSE;
    			Delay_TON6();
    			Motor6.Seq := 3;
    		END_IF;
    			
    	3 : // 원점까지 Motor 정방향 회전
    		IF NOT FB_Motor6_Control.Done AND NOT Sensor6_L THEN
    			Motor6Control.TargetPulse := 20000;
    			Motor6Control.SetDir	:= FALSE;
    			Motor6Control.MoveStart := TRUE;
    		ELSE
    			Motor6Control.MoveStart := FALSE;
    			Motor6.Seq := 7;
    		END_IF;
    		
    	4: // Motor 
    		IF NOT FB_Motor6_Control.Done AND NOT Sensor6_L THEN
    			Motor6Control.TargetPulse := 1375;
    			Motor6Control.SetDir := FALSE;
    			Motor6Control.MoveStart:=TRUE;
    		END_IF;
    		
    		IF FB_Motor6_Control.Done THEN
    			Motor6Control.MoveStart := FALSE;
    			Motor6.Seq := 0;
    		END_IF;
    		
    	5: // Motor 
    		IF NOT FB_Motor6_Control.Done AND NOT Sensor6_R THEN
    			Motor6Control.TargetPulse := 1375;
    			Motor6Control.SetDir := TRUE;
    			Motor6Control.MoveStart:=TRUE;
    		END_IF;
    		
    		IF FB_Motor6_Control.Done THEN
    			Motor6Control.MoveStart := FALSE;
    			Motor6.Seq := 0;
    		END_IF;
    	
    	6: // 지정 거리 이동
    		IF NOT FB_Motor6_Control.Done AND NOT Sensor6_L AND NOT Sensor6_R THEN
    			IF Motor6.Move >= 0 THEN
    				Motor6Control.SetDir := TRUE;
    			ELSIF Motor6.Move < 0 THEN
    				Motor6Control.SetDir := FALSE;
    			END_IF;
    			
    			Motor6Control.TargetPulse := ABS(Motor6.Move)*200/80;
    			Motor6Control.MoveStart := TRUE;
    			Finish6:=FALSE;
    		END_IF;
    		
    		IF FB_Motor6_Control.Done THEN
    			Motor6Control.MoveStart := FALSE;
    			Finish6:=TRUE;
    			Motor6.Seq := 0;
    		END_IF;
    	
    	7: // LSL 도달 시 복귀
    		IF NOT FB_Motor6_Control.Done AND Sensor6_L THEN
    			Motor6Control.TargetPulse := 193;
    			Motor6Control.SetDir := TRUE;
    			Motor6Control.MoveStart := TRUE;
    		END_IF;
    		
    		IF FB_Motor6_Control.Done THEN
    			Motor6Control.MoveStart := FALSE;
    			Finish6:=TRUE;
    			Motor6.Seq := 0;
    		END_IF;
    		
    	8: // RSL 도달 시 복귀
    		IF NOT FB_Motor6_Control.Done AND Sensor6_R THEN
    			Motor6Control.TargetPulse := 180;
    			Motor6Control.SetDir := FALSE;
    			Motor6Control.MoveStart := TRUE;
    		END_IF;
    		
    		IF FB_Motor6_Control.Done THEN
    			Motor6Control.MoveStart := FALSE;
    			Motor6.Seq := 0;
    		END_IF;
    END_CASE;
END_IF;

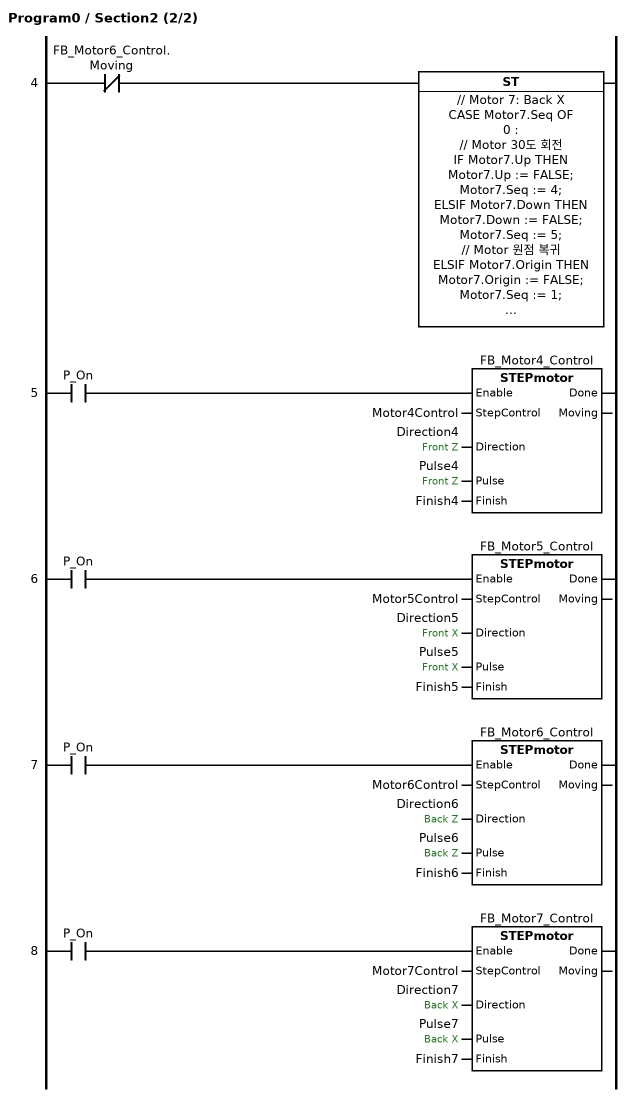
(* Rung 4 *)
IF NOT FB_Motor6_Control.Moving THEN
    // Motor 7: Back X
    	
    CASE Motor7.Seq OF
    	
    	0 : 
    		// Motor 30도 회전
    		IF Motor7.Up THEN
    			Motor7.Up := FALSE;
    			Motor7.Seq := 4;
    		ELSIF Motor7.Down THEN
    			Motor7.Down := FALSE;
    			Motor7.Seq := 5;
    		// Motor 원점 복귀
    		ELSIF Motor7.Origin THEN
    			Motor7.Origin := FALSE;
    			Motor7.Seq := 1;
    		// Motor.Check 가 TRUE 면 Motor.Move 에 설정된 거리만큼 이동
    		ELSIF Motor7.Check THEN
    			Motor7.Check := FALSE;
    			Motor7.Seq := 6;
    		
    		END_IF;
    		
    		
    	1 : // Motor 15도 역방향 회전
    		IF NOT FB_Motor7_Control.Done 
    			AND NOT Sensor7_L 
    			AND NOT Sensor7_R THEN
    			Motor7Control.TargetPulse := 50;
    			Motor7Control.SetDir	:= TRUE;
    			Motor7Control.MoveStart := TRUE;
    			Finish7:=FALSE;
    		END_IF;
    		
    		IF FB_Motor7_Control.Done THEN
    			Motor7Control.MoveStart := FALSE;
    			Motor7.Seq := 2;
    		END_IF;
    		
    	2: // 0.5s delay
    		Delay_TON7.In := TRUE;
    		Delay_TON7.PT := T#0.5s;
    		Delay_TON7();
    		
    		IF Delay_TON7.Q THEN
    			Delay_TON7.In := FALSE;
    			Delay_TON7();
    			Motor7.Seq := 3;
    		END_IF;
    			
    	3 : // 원점까지 Motor 정방향 회전
    		IF NOT FB_Motor7_Control.Done AND NOT Sensor7_L THEN
    			Motor7Control.TargetPulse := 20000;
    			Motor7Control.SetDir	:= FALSE;
    			Motor7Control.MoveStart := TRUE;
    		ELSE
    			Motor7Control.MoveStart := FALSE;
    			Motor7.Seq := 7;
    		END_IF;
    		
    	4: // Motor 
    		IF NOT FB_Motor7_Control.Done AND NOT Sensor7_L THEN
    			Motor7Control.TargetPulse := 900;
    			Motor7Control.SetDir := TRUE;
    			Motor7Control.MoveStart:=TRUE;
    		END_IF;
    		
    		IF FB_Motor7_Control.Done THEN
    			Motor7Control.MoveStart := FALSE;
    			Motor7.Seq := 0;
    		END_IF;
    		
    	5: // Motor 
    		IF NOT FB_Motor7_Control.Done AND NOT Sensor7_R THEN
    			Motor7Control.TargetPulse := 900;
    			Motor7Control.SetDir := FALSE;
    			Motor7Control.MoveStart:=TRUE;
    		END_IF;
    		
    		IF FB_Motor7_Control.Done THEN
    			Motor7Control.MoveStart := FALSE;
    			Motor7.Seq := 0;
    		END_IF;
    	
    	6: // 지정 거리 이동
    		IF NOT FB_Motor7_Control.Done AND NOT Sensor7_L AND NOT Sensor7_R THEN
    			IF Motor7.Move >= 0 THEN
    				Motor7Control.SetDir := TRUE;
    			ELSIF Motor7.Move < 0 THEN
    				Motor7Control.SetDir := FALSE;
    			END_IF;
    			
    			Motor7Control.TargetPulse := ABS(Motor7.Move)*200/100;
    			Motor7Control.MoveStart := TRUE;
    			Finish7:=FALSE;
    		END_IF;
    		
    		IF FB_Motor7_Control.Done THEN
    			Motor7Control.MoveStart := FALSE;
    			Finish7:=TRUE;
    			Motor7.Seq := 0;
    		END_IF;
    	
    	7: // LSL 도달 시 복귀
    		IF NOT FB_Motor7_Control.Done AND Sensor7_L THEN
    			Motor7Control.TargetPulse := 240;
    			Motor7Control.SetDir := TRUE;
    			Motor7Control.MoveStart := TRUE;
    		END_IF;
    		
    		IF FB_Motor7_Control.Done THEN
    			Motor7Control.MoveStart := FALSE;
    			Finish7:=TRUE;
    			Motor7.Seq := 0;
    		END_IF;
    		
    		8: // RSL 도달 시 복귀
    		IF NOT FB_Motor7_Control.Done AND Sensor7_R THEN
    			Motor7Control.TargetPulse := 180;
    			Motor7Control.SetDir := FALSE;
    			Motor7Control.MoveStart := TRUE;
    		END_IF;
    		
    		IF FB_Motor7_Control.Done THEN
    			Motor7Control.MoveStart := FALSE;
    			Motor7.Seq := 0;
    		END_IF;
    END_CASE;
END_IF;
(* Rung 5 *)
FB_Motor4_Control(Enable := P_On, StepControl := Motor4Control, Direction := Direction4, Pulse := Pulse4, Finish := Finish4);
(* Rung 6 *)
FB_Motor5_Control(Enable := P_On, StepControl := Motor5Control, Direction := Direction5, Pulse := Pulse5, Finish := Finish5);
(* Rung 7 *)
FB_Motor6_Control(Enable := P_On, StepControl := Motor6Control, Direction := Direction6, Pulse := Pulse6, Finish := Finish6);
(* Rung 8 *)
FB_Motor7_Control(Enable := P_On, StepControl := Motor7Control, Direction := Direction7, Pulse := Pulse7, Finish := Finish7);

(* Section Section3: ladder, written here as Structured Text *)

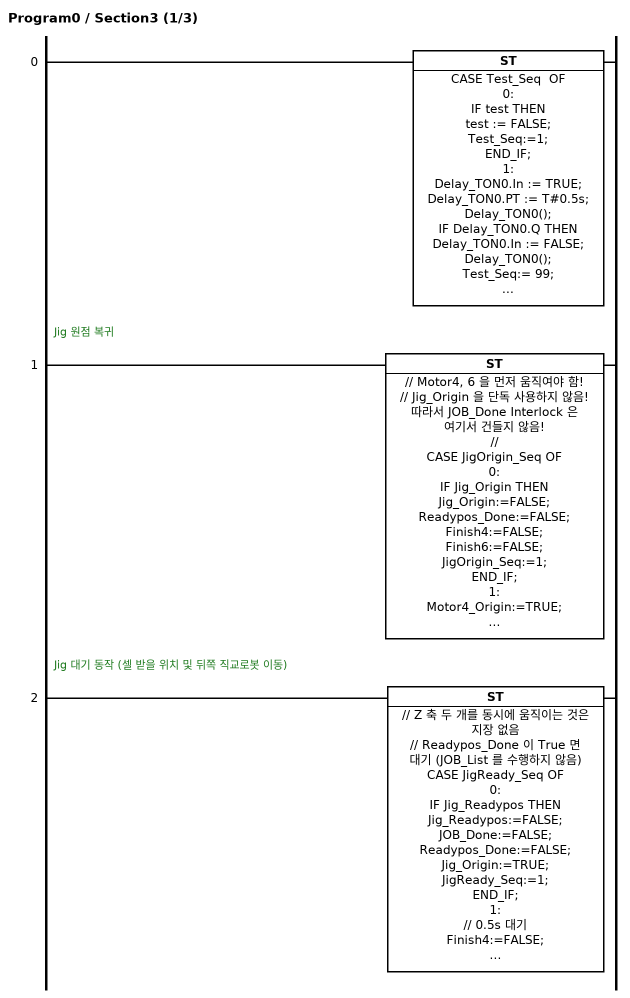
(* Rung 0 *)
CASE Test_Seq  OF
	0:
		IF test THEN
			test := FALSE;
			Test_Seq:=1;
		END_IF;
	1:
		Delay_TON0.In := TRUE;
		Delay_TON0.PT := T#0.5s;
		Delay_TON0();
			
		IF Delay_TON0.Q THEN
			Delay_TON0.In := FALSE;
			Delay_TON0();
			Test_Seq:= 99;
		END_IF;
	99:
		Delay_TON0.In := TRUE;
		Delay_TON0.PT := T#0.5s;
		Delay_TON0();
			
		IF Delay_TON0.Q THEN
			Delay_TON0.In := FALSE;
			Delay_TON0();
			Test_Seq:= 0;
		END_IF;
END_CASE;
(* Rung 1: Jig 원점 복귀 *)
// Motor4, 6 을 먼저 움직여야 함!
// Jig_Origin 을 단독 사용하지 않음! 따라서 JOB_Done Interlock 은 여기서 건들지 않음!
//
CASE JigOrigin_Seq OF
	0:
		IF Jig_Origin THEN
			Jig_Origin:=FALSE;
			Readypos_Done:=FALSE;
			Finish4:=FALSE;
			Finish6:=FALSE;
			JigOrigin_Seq:=1;
		END_IF;
		
	1:
		Motor4_Origin:=TRUE;
		Motor6_Origin:=TRUE;
		Finish5:=FALSE;
		Finish7:=FALSE;
		JigOrigin_Seq:= 2;
		
	2:
		Delay_TON8.In := TRUE;
		Delay_TON8.PT := T#0.5s;
		Delay_TON8();
			
		IF Delay_TON8.Q THEN
			Delay_TON8.In := FALSE;
			Delay_TON8();
			JigOrigin_Seq:= 3;
		END_IF;
		
	3:
		IF Finish4 	AND Finish6 THEN
			Motor5_Origin:=TRUE;
			Motor7_Origin:=TRUE;
			JigOrigin_Seq:=0;
		END_IF;
		
END_CASE;
(* Rung 2: Jig 대기 동작 (셀 받을 위치 및 뒤쪽 직교로봇 이동) *)
// Z 축 두 개를 동시에 움직이는 것은 지장 없음
// Readypos_Done 이 True 면 대기 (JOB_List 를 수행하지 않음)
CASE JigReady_Seq OF
	0:
		IF Jig_Readypos THEN
			Jig_Readypos:=FALSE;
			JOB_Done:=FALSE;
			Readypos_Done:=FALSE;
			Jig_Origin:=TRUE;
			JigReady_Seq:=1;
		END_IF;
	
	1:
		// 0.5s 대기
		Finish4:=FALSE;
		
		Delay_TON9.In := TRUE;
		Delay_TON9.PT := T#0.5s;
		Delay_TON9();
		
		IF Delay_TON9.Q THEN
			Delay_TON9.In := FALSE;
			Delay_TON9();
			JigReady_Seq:= 2;
		END_IF;
		
	2:
		IF NOT JOB_Done AND Finish5 AND Finish7 THEN
			Motor4_Move:=430;
			Motor7_Move:=400;
			Motor4_Check:=TRUE;
			Motor7_Check:=TRUE;
			JigReady_Seq:=3;
		END_IF;
		
	3:
		IF Finish4 THEN
			JOB_Done:=TRUE;
			Readypos_Done:=TRUE;
			JigReady_Seq:=0;
		END_IF;
		
END_CASE;

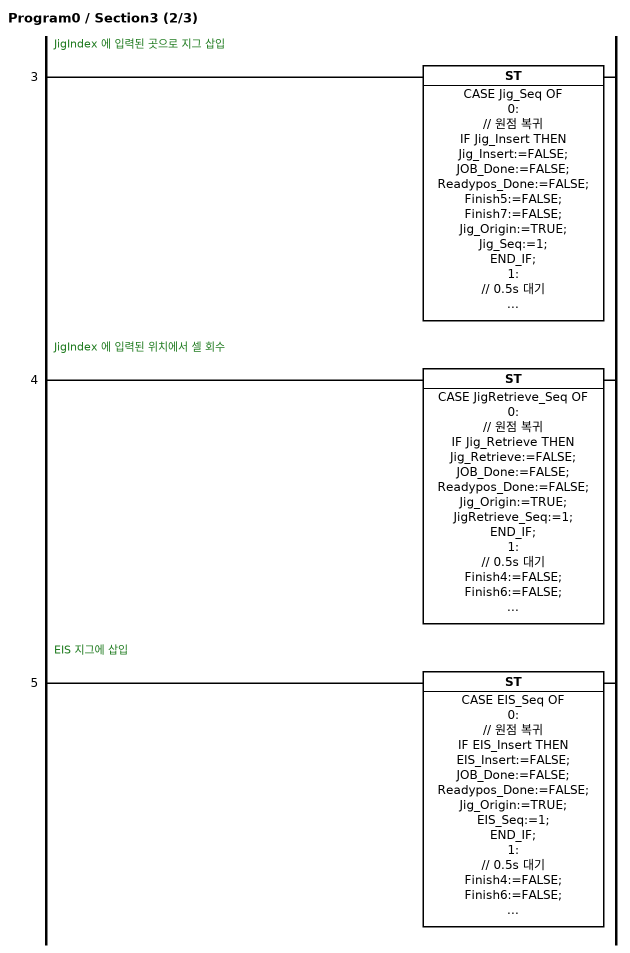
(* Rung 3: JigIndex 에 입력된 곳으로 지그 삽입 *)
CASE Jig_Seq OF
	0:
		// 원점 복귀
		IF Jig_Insert THEN
			Jig_Insert:=FALSE;
			JOB_Done:=FALSE;
			Readypos_Done:=FALSE;
			
			Finish5:=FALSE;
			Finish7:=FALSE;
			Jig_Origin:=TRUE;
			Jig_Seq:=1;
		END_IF;
	
	1: 
		// 0.5s 대기
		Delay_TON10.In := TRUE;
		Delay_TON10.PT := T#0.5s;
		Delay_TON10();
		
		IF Delay_TON10.Q THEN
			Delay_TON10.In := FALSE;
			Delay_TON10();
			Jig_Seq:= 2;
		END_IF;
		
	2:
		// X 축 이동 (앞쪽 모터는 225 만큼 빼서)
		IF NOT JOB_Done AND Finish5 AND Finish7 THEN
			Finish5:=FALSE;
			Finish7:=FALSE;
			Motor5_Move:=TO_INT(Jigmove_csv[JigIndex,1]*10.0)-225;
			Motor7_Move:=TO_INT(Jigmove_csv[JigIndex,5]*10.0);
			Motor5_Check:=TRUE;
			Motor7_Check:=TRUE;
			Jig_Seq:=3;
		END_IF;
		
		
	3:
		// 0.5s 대기
		Delay_TON10.In := TRUE;
		Delay_TON10.PT := T#0.5s;
		Delay_TON10();
		
		IF Delay_TON10.Q THEN
			Delay_TON10.In := FALSE;
			Delay_TON10();
			Jig_Seq:= 4;
		END_IF;
		
	4:
		// Z 축 이동
		IF Finish5 AND Finish7 THEN
			Finish4:=FALSE;
			Finish6:=FALSE;
			Motor4_Move:=TO_INT(Jigmove_csv[JigIndex,0]*10.0);
			Motor6_Move:=TO_INT(Jigmove_csv[JigIndex,4]*10.0);
			Motor4_Check:=TRUE;
			Motor6_Check:=TRUE;
			Jig_Seq:=5;
		END_IF;
		
	5:
		//0.5s 대기
		Delay_TON10.In := TRUE;
		Delay_TON10.PT := T#0.5s;
		Delay_TON10();
		
		IF Delay_TON10.Q THEN
			Delay_TON10.In := FALSE;
			Delay_TON10();
			Jig_Seq:= 6;
		END_IF;
		
	6:
		// 액츄 지그 오른쪽으로 약간 이동
		IF Finish4 AND Finish6 THEN
			Finish5:=FALSE;
			Motor5_Move:=225;
			Motor5_Check:=TRUE;
			Jig_Seq:=7;
		END_IF;
		
	7:
		//0.5s 대기
		Delay_TON10.In := TRUE;
		Delay_TON10.PT := T#0.5s;
		Delay_TON10();
		
		IF Delay_TON10.Q THEN
			Delay_TON10.In := FALSE;
			Delay_TON10();
			Jig_Seq:= 8;
		END_IF;
	
	8: 
		// 지그 개방 (Motor7 먼저 움직여야 함)
		IF Finish5 THEN
			Finish7:=FALSE;
			Motor7_Move:=225;
			Motor7_Check:=TRUE;
			Jig_Seq:=9;
		END_IF;
		
	9:
		// 0.5s 대기
		Delay_TON10.In := TRUE;
		Delay_TON10.PT := T#0.5s;
		Delay_TON10();
		
		IF Delay_TON10.Q THEN
			Delay_TON10.In := FALSE;
			Delay_TON10();
			Jig_Seq:= 10;
		END_IF;
		
	10:
		// 지그 개방 (Motor6 움직임)
		IF Finish7 THEN
			Finish6:=FALSE;
			Motor6_Move:=120;
			Motor6_Check:=TRUE;
			Jig_Seq:=11;
		END_IF;
		
	11:
		// 0.5s 대기
		Delay_TON10.In := TRUE;
		Delay_TON10.PT := T#0.5s;
		Delay_TON10();
		
		IF Delay_TON10.Q THEN
			Delay_TON10.In := FALSE;
			Delay_TON10();
			Jig_Seq:= 12;
		END_IF;
		
	12:
		// 액츄에이터 삽입
		IF Finish6 THEN
			ActuIndex:=13;
			ActuMove:=TO_INT(Jigmove_csv[JigIndex,2]);
			Open_Serial:=TRUE;
			Jig_Seq:=13;
		END_IF;
		
	13:
		// 액츄에이터 통신 종료 확인 및 0.5s 기다림		
		IF NOT Serial_Busy THEN
			Delay_TON10.In := TRUE;
			Delay_TON10.PT := T#1s;
			Delay_TON10();
			
			IF Delay_TON10.Q THEN
				Delay_TON10.In := FALSE;
				Delay_TON10();
				Jig_Seq:= 14;
			END_IF;
		END_IF;
	
	14:
		// 지그 닫음 (Motor6 먼저 움직여야 함!)
		Finish6:=FALSE;
		Motor6_Move:=-120;
		Motor6_Check:=TRUE;
		Jig_Seq:=15;
		
	15:
		// 0.5s 대기
		Delay_TON10.In := TRUE;
		Delay_TON10.PT := T#0.5s;
		Delay_TON10();
		
		IF Delay_TON10.Q THEN
			Delay_TON10.In := FALSE;
			Delay_TON10();
			Jig_Seq:= 16;
		END_IF;
		
	16:
		// 지그 닫음 (Motor7 움직임)
		IF Finish6 THEN
			Finish7:=FALSE;
			Motor7_Move:=-225;
			Motor7_Check:=TRUE;
			Jig_Seq:=17;
		END_IF;
	
	17:
		// 0,5s 대기
		Delay_TON10.In := TRUE;
		Delay_TON10.PT := T#0.5s;
		Delay_TON10();
		
		IF Delay_TON10.Q THEN
			Delay_TON10.In := FALSE;
			Delay_TON10();
			Jig_Seq:= 18;
		END_IF;
		
	18:
		// 액츄에이터 지그 하강
		IF Finish7 THEN;
			Finish4:=FALSE;
			Motor4_Move:=TO_INT(Jigmove_csv[JigIndex,3]*10.0);
			Motor4_Check:=TRUE;
			Jig_Seq:=19;
		END_IF;
		
	19:
		// 0,5s 대기
		Delay_TON10.In := TRUE;
		Delay_TON10.PT := T#0.5s;
		Delay_TON10();
		
		IF Delay_TON10.Q THEN
			Delay_TON10.In := FALSE;
			Delay_TON10();
			Jig_Seq:= 20;
		END_IF;
	
	20:
		// 액츄에이터 후진
		IF Finish4 THEN
			ActuIndex:=13;
			ActuMove:=0;
			Open_Serial:=TRUE;
			Jig_Seq:=21;
		END_IF;
		
	21:
		// 액츄에이터 통신 종료 확인 및  0,5s 대기
		// Finish5:=FALSE;
		// Finish7:=FALSE;
		
		IF NOT Serial_Busy THEN
			Delay_TON10.In := TRUE;
			Delay_TON10.PT := T#1s;
			Delay_TON10();
			
			IF Delay_TON10.Q THEN
				Delay_TON10.In := FALSE;
				Delay_TON10();
				Jig_Seq:= 22;
			END_IF;
		END_IF;
		
	22:
		// 원점 복귀
		Finish5:=FALSE;
		Finish7:=FALSE;
		
		Jig_Origin:=TRUE;
		Jig_Seq:=23;
		
	23:
		IF Finish5 AND Finish7 THEN
			JOB_Done:=TRUE;
			Jig_Seq:=0;
		END_IF;

END_CASE;
(* Rung 4: JigIndex 에 입력된 위치에서 셀 회수 *)
CASE JigRetrieve_Seq OF
	0:
		// 원점 복귀
		IF Jig_Retrieve THEN
			Jig_Retrieve:=FALSE;
			JOB_Done:=FALSE;
			Readypos_Done:=FALSE;
			Jig_Origin:=TRUE;
			JigRetrieve_Seq:=1;
		END_IF;
	
	1: 
		// 0.5s 대기
		Finish4:=FALSE;
		Finish6:=FALSE;
		
		Delay_TON11.In := TRUE;
		Delay_TON11.PT := T#0.5s;
		Delay_TON11();
		
		IF Delay_TON11.Q THEN
			Delay_TON11.In := FALSE;
			Delay_TON11();
			JigRetrieve_Seq:= 2;
		END_IF;
		
	2:
		// Z 축 이동
		IF NOT JOB_Done AND Finish5 AND Finish7 THEN
			Motor4_Move:=TO_INT(Jigmove_csv[JigIndex,0]*10.0);
			Motor6_Move:=TO_INT(Jigmove_csv[JigIndex,4]*10.0);
			Motor4_Check:=TRUE;
			Motor6_Check:=TRUE;
			JigRetrieve_Seq:=3;
		END_IF;
		
		
	3:
		// 0.5s 대기
		Finish5:=FALSE;
		Finish7:=FALSE;
		
		Delay_TON11.In := TRUE;
		Delay_TON11.PT := T#0.5s;
		Delay_TON11();
		
		IF Delay_TON11.Q THEN
			Delay_TON11.In := FALSE;
			Delay_TON11();
			JigRetrieve_Seq:= 4;
		END_IF;
		
	4:
		// X 축 이동
		IF Finish4 AND Finish6 THEN
			Motor5_Move:=TO_INT(Jigmove_csv[JigIndex,1]*10.0);
			Motor7_Move:=TO_INT(Jigmove_csv[JigIndex,5]*10.0);
			Motor5_Check:=TRUE;
			Motor7_Check:=TRUE;
			JigRetrieve_Seq:=5;
		END_IF;
		
	5:
		//0.5s 대기
		Finish4:=FALSE;
		
		Delay_TON11.In := TRUE;
		Delay_TON11.PT := T#0.5s;
		Delay_TON11();
		
		IF Delay_TON11.Q THEN
			Delay_TON11.In := FALSE;
			Delay_TON11();
			JigRetrieve_Seq:= 6;
		END_IF;
	
	6: 
		// 액츄에이터 지그 하강
		IF Finish7 THEN;
			Motor4_Move:=TO_INT(Jigmove_csv[JigIndex,3]*10.0);
			Motor4_Check:=TRUE;
			JigRetrieve_Seq:=7;
		END_IF;
		
	7:
		// 0.5s 대기		
		Delay_TON11.In := TRUE;
		Delay_TON11.PT := T#0.5s;
		Delay_TON11();
		
		IF Delay_TON11.Q THEN
			Delay_TON11.In := FALSE;
			Delay_TON11();
			JigRetrieve_Seq:= 8;
		END_IF;
		
	8:
		// 액츄에이터 삽입
		IF Finish4 THEN
			ActuIndex:=13;
			ActuMove:=TO_INT(Jigmove_csv[JigIndex,2]);
			Open_Serial:=TRUE;
			JigRetrieve_Seq:=9;
		END_IF;
		
	9:
		// 액츄에이터 통신 종료 확인 및 0.5s 기다림
		Finish7:=FALSE;
		
		IF NOT Serial_Busy THEN
			Delay_TON11.In := TRUE;
			Delay_TON11.PT := T#1s;
			Delay_TON11();
			
			IF Delay_TON11.Q THEN
				Delay_TON11.In := FALSE;
				Delay_TON11();
				JigRetrieve_Seq:= 10;
			END_IF;
		END_IF;
		
	10:
		// 지그 개방 (Motor7 먼저 움직여야 함)
		Motor7_Move:=225;
		Motor7_Check:=TRUE;
		JigRetrieve_Seq:=11;
		
	11:
		// 0.5s 대기
		Finish6:=FALSE;
		
		Delay_TON11.In := TRUE;
		Delay_TON11.PT := T#0.5s;
		Delay_TON11();
		
		IF Delay_TON11.Q THEN
			Delay_TON11.In := FALSE;
			Delay_TON11();
			JigRetrieve_Seq:= 12;
		END_IF;
		
	12:
		// 지그 개방 (Motor6 움직임)
		IF Finish7 THEN
			Motor6_Move:=120;
			Motor6_Check:=TRUE;
			JigRetrieve_Seq:=13;
		END_IF;
	
	13:
		// 0.5s 대기
		Finish4:=FALSE;
		
		Delay_TON11.In := TRUE;
		Delay_TON11.PT := T#0.5s;
		Delay_TON11();
		
		IF Delay_TON11.Q THEN
			Delay_TON11.In := FALSE;
			Delay_TON11();
			JigRetrieve_Seq:= 14;
		END_IF;
		
	14:
		// 액츄에이터 지그 상승
		IF Finish6 THEN;
			Motor4_Move:=-TO_INT(Jigmove_csv[JigIndex,3]*10.0);
			Motor4_Check:=TRUE;
			JigRetrieve_Seq:=15;
		END_IF;
	
	15:
		// 0,5s 대기
		Delay_TON11.In := TRUE;
		Delay_TON11.PT := T#0.5s;
		Delay_TON11();
		
		IF Delay_TON11.Q THEN
			Delay_TON11.In := FALSE;
			Delay_TON11();
			JigRetrieve_Seq:= 16;
		END_IF;
		
	16:
		// 액츄에이터 후진
		IF Finish4 THEN
			ActuIndex:=13;
			ActuMove:=0;
			Open_Serial:=TRUE;
			JigRetrieve_Seq:=17;
		END_IF;
		
	17:
		// 액츄에이터 통신 종료 확인 및 0.5s 기다림
		Finish6:=FALSE;
		
		IF NOT Serial_Busy THEN
			Delay_TON11.In := TRUE;
			Delay_TON11.PT := T#1s;
			Delay_TON11();
			
			IF Delay_TON11.Q THEN
				Delay_TON11.In := FALSE;
				Delay_TON11();
				JigRetrieve_Seq:= 18;
			END_IF;
		END_IF;
	
	18:
		// 지그 닫음 (Motor6 먼저 움직여야 함!)
		Motor6_Move:=-120;
		Motor6_Check:=TRUE;
		JigRetrieve_Seq:=19;
		
	19:
		// 0,5s 대기
		Finish7:=FALSE;
		
		Delay_TON11.In := TRUE;
		Delay_TON11.PT := T#0.5s;
		Delay_TON11();
		
		IF Delay_TON11.Q THEN
			Delay_TON11.In := FALSE;
			Delay_TON11();
			JigRetrieve_Seq:= 20;
		END_IF;
		
	20:
		// 지그 닫음 (Motor7 움직임)
		IF Finish6 THEN
			Motor7_Move:=-225;
			Motor7_Check:=TRUE;
			JigRetrieve_Seq:=21;
		END_IF;
		
	21:
		// 0,5s 대기
		Finish5:=FALSE;
		
		Delay_TON11.In := TRUE;
		Delay_TON11.PT := T#0.5s;
		Delay_TON11();
		
		IF Delay_TON11.Q THEN
			Delay_TON11.In := FALSE;
			Delay_TON11();
			JigRetrieve_Seq:= 22;
		END_IF;
		
	22:
		// 액츄 지그 왼쪽으로 약간 이동
		IF Finish7 THEN
			Motor5_Move:=-225;
			Motor5_Check:=TRUE;
			JigRetrieve_Seq:=23;
		END_IF;
	
	23:
		// 0,5s 대기
		Delay_TON11.In := TRUE;
		Delay_TON11.PT := T#0.5s;
		Delay_TON11();
		
		IF Delay_TON11.Q THEN
			Delay_TON11.In := FALSE;
			Delay_TON11();
			JigRetrieve_Seq:= 24;
		END_IF;
		
	24:
		// 원점 복귀
		IF Finish5 THEN
			Finish5:=FALSE;
			Finish7:=FALSE;
			Jig_Origin:=TRUE;
			JigRetrieve_Seq:=25;
		END_IF;
		
	25:
		IF Finish5 AND Finish7 THEN
			JOB_Done:=TRUE;
			JigRetrieve_Seq:=0;
		END_IF;

END_CASE;
(* Rung 5: EIS 지그에 삽입 *)
CASE EIS_Seq OF
	0:
		// 원점 복귀
		IF EIS_Insert THEN
			EIS_Insert:=FALSE;
			JOB_Done:=FALSE;
			Readypos_Done:=FALSE;
			Jig_Origin:=TRUE;
			EIS_Seq:=1;
		END_IF;
	
	1: 
		// 0.5s 대기
		Finish4:=FALSE;
		Finish6:=FALSE;
		
		Delay_TON12.In := TRUE;
		Delay_TON12.PT := T#0.5s;
		Delay_TON12();
		
		IF Delay_TON12.Q THEN
			Delay_TON12.In := FALSE;
			Delay_TON12();
			EIS_Seq:= 2;
		END_IF;
		
	2:
		// Z 축 이동
		IF NOT JOB_Done AND Finish5 AND Finish7 THEN
			Motor4_Move:=TO_INT(EISmove_csv[EISIndex,0]*10.0);
			Motor6_Move:=TO_INT(EISmove_csv[EISIndex,0]*10.0);
			Motor4_Check:=TRUE;
			Motor6_Check:=TRUE;
			EIS_Seq:=3;
		END_IF;
		
		
	3:
		// 0.5s 대기
		Finish5:=FALSE;
		
		Delay_TON12.In := TRUE;
		Delay_TON12.PT := T#0.5s;
		Delay_TON12();
		
		IF Delay_TON12.Q THEN
			Delay_TON12.In := FALSE;
			Delay_TON12();
			EIS_Seq:= 4;
		END_IF;
		
	4:
		// X 축 이동
		IF Finish4 THEN
			Motor5_Move:=TO_INT(EISmove_csv[EISIndex,1]*10.0);
			Motor5_Check:=TRUE;
			EIS_Seq:=5;
		END_IF;
		
	5:
		//0.5s 대기
		Delay_TON12.In := TRUE;
		Delay_TON12.PT := T#0.5s;
		Delay_TON12();
		
		IF Delay_TON12.Q THEN
			Delay_TON12.In := FALSE;
			Delay_TON12();
			EIS_Seq:= 6;
		END_IF;
	
	6: 
		// 지그 개방 (액츄에이터 기동)
		IF Finish5 THEN
			IF EISIndex = 0 THEN
				ActuIndex:=12;
				ActuMove:=TO_INT(EISmove_csv[EISIndex,3]);
				Open_Serial:=TRUE;
				EIS_Seq:=7;
			ELSIF EISIndex=1 THEN
				ActuIndex:=11;
				ActuMove:=TO_INT(EISmove_csv[EISIndex,3]);
				Open_Serial:=TRUE;
				EIS_Seq:=7;
			END_IF;
		END_IF;
		
	7:
		// 액츄에이터 통신 종료 확인 및 0.5s 기다림
		IF NOT Serial_Busy THEN
			Delay_TON12.In := TRUE;
			Delay_TON12.PT := T#1s;
			Delay_TON12();
			
			IF Delay_TON12.Q THEN
				Delay_TON12.In := FALSE;
				Delay_TON12();
				EIS_Seq:= 8;
			END_IF;
		END_IF;
		
	8:
		// 액츄에이터 삽입
		ActuIndex:=13;
		ActuMove:=TO_INT(EISmove_csv[EISIndex,2]);
		Open_Serial:=TRUE;
		EIS_Seq:=9;
		
	9:
		// 액츄에이터 통신 종료 확인 및 0.5s 기다림
		IF NOT Serial_Busy THEN
			Delay_TON12.In := TRUE;
			Delay_TON12.PT := T#1s;
			Delay_TON12();
			
			IF Delay_TON12.Q THEN
				Delay_TON12.In := FALSE;
				Delay_TON12();
				EIS_Seq:= 10;
			END_IF;
		END_IF;
		
	10:
		// 지그 폐쇄 (액츄에이터 기동)
		IF EISIndex = 0 THEN
			ActuIndex:=12;
		ELSIF EISIndex=1 THEN
			ActuIndex:=11;
		END_IF;
		ActuMove:=0;
		Open_Serial:=TRUE;
		EIS_Seq:=11;
		
	11:
		// 액츄에이터 통신 종료 확인 및 0.5s 기다림
		IF NOT Serial_Busy THEN
			Delay_TON12.In := TRUE;
			Delay_TON12.PT := T#1s;
			Delay_TON12();
			
			IF Delay_TON12.Q THEN
				Delay_TON12.In := FALSE;
				Delay_TON12();
				EIS_Seq:= 12;
			END_IF;
		END_IF;
	
	12:
		// 액츄에이터 회수
		ActuIndex:=13;
		ActuMove:=0;
		Open_Serial:=TRUE;		
		EIS_Seq:=13;
		
	13:
		// 액츄에이터 통신 종료 확인 및 0.5s 기다림
		Finish5:=FALSE;
		
		IF NOT Serial_Busy THEN
			Delay_TON12.In := TRUE;
			Delay_TON12.PT := T#1s;
			Delay_TON12();
			
			IF Delay_TON12.Q THEN
				Delay_TON12.In := FALSE;
				Delay_TON12();
				EIS_Seq:= 14;
			END_IF;
		END_IF;
	
	14:
		// 왼쪽으로 이동
		IF EISIndex=0 THEN
			Motor5_Move:=-850;
			Motor5_Check:=TRUE;
			EIS_Seq:=15;
		ELSIF EISIndex=1 THEN
			Motor5_Move:=-1250;
			Motor5_Check:=TRUE;
			EIS_Seq:=15;
		END_IF;
		
	15:
		// 0.5s 대기
		Delay_TON12.In := TRUE;
		Delay_TON12.PT := T#0.5s;
		Delay_TON12();
		
		IF Delay_TON12.Q THEN
			Delay_TON12.In := FALSE;
			Delay_TON12();
			EIS_Seq:= 16;
		END_IF;
		
	16:
		// 원점 복귀
		IF Finish5 THEN
			Finish5:=FALSE;
			Finish7:=FALSE;
			Jig_Origin:=TRUE;
			EIS_Seq:=17;
		END_IF;
		
	17:
		IF Finish5 AND Finish7 THEN
			JOB_Done:=TRUE;
			EIS_Seq:=0;
		END_IF;

END_CASE;

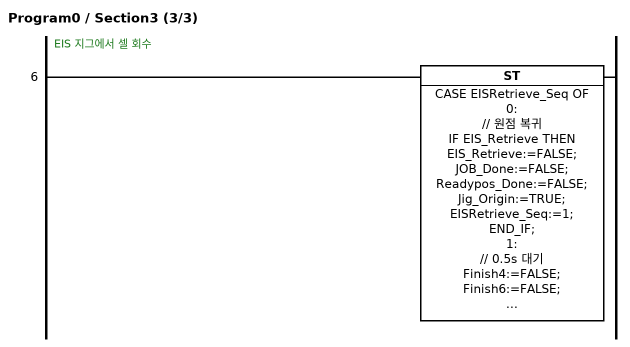
(* Rung 6: EIS 지그에서 셀 회수 *)
CASE EISRetrieve_Seq OF
	0:
		// 원점 복귀
		IF EIS_Retrieve THEN
			EIS_Retrieve:=FALSE;
			JOB_Done:=FALSE;
			Readypos_Done:=FALSE;
			Jig_Origin:=TRUE;
			EISRetrieve_Seq:=1;
		END_IF;
	
	1: 
		// 0.5s 대기
		Finish4:=FALSE;
		Finish6:=FALSE;
		
		Delay_TON13.In := TRUE;
		Delay_TON13.PT := T#0.5s;
		Delay_TON13();
		
		IF Delay_TON13.Q THEN
			Delay_TON13.In := FALSE;
			Delay_TON13();
			EISRetrieve_Seq:= 2;
		END_IF;
		
	2:
		// Z 축 이동
		IF NOT JOB_Done AND Finish5 AND Finish7 THEN
			Motor4_Move:=TO_INT(EISmove_csv[EISIndex,0]*10.0);
			Motor6_Move:=TO_INT(EISmove_csv[EISIndex,0]*10.0);
			Motor4_Check:=TRUE;
			Motor6_Check:=TRUE;
			EISRetrieve_Seq:=3;
		END_IF;
		
		
	3:
		// 0.5s 대기
		Finish5:=FALSE;
		
		Delay_TON13.In := TRUE;
		Delay_TON13.PT := T#0.5s;
		Delay_TON13();
		
		IF Delay_TON13.Q THEN
			Delay_TON13.In := FALSE;
			Delay_TON13();
			EISRetrieve_Seq:= 4;
		END_IF;
		
	4:
		// X 축 이동
		IF Finish4 THEN
			Motor5_Move:=TO_INT(EISmove_csv[EISIndex,1]*10.0);
			Motor5_Check:=TRUE;
			EISRetrieve_Seq:=5;
		END_IF;
		
	5:
		//0.5s 대기
		Delay_TON13.In := TRUE;
		Delay_TON13.PT := T#0.5s;
		Delay_TON13();
		
		IF Delay_TON13.Q THEN
			Delay_TON13.In := FALSE;
			Delay_TON13();
			EISRetrieve_Seq:= 6;
		END_IF;
	
	6: 
		// 액츄에이터 삽입
		IF Finish5 THEN
		ActuIndex:=13;
		ActuMove:=TO_INT(EISmove_csv[EISIndex,2]);
		Open_Serial:=TRUE;
		EISRetrieve_Seq:=7;
		END_IF;
		
	7:
		// 액츄에이터 통신 종료 확인 및 3s 기다림
		IF NOT Serial_Busy THEN
			Delay_TON13.In := TRUE;
			Delay_TON13.PT := T#1s;
			Delay_TON13();
			
			IF Delay_TON13.Q THEN
				Delay_TON13.In := FALSE;
				Delay_TON13();
				EISRetrieve_Seq:= 8;
			END_IF;
		END_IF;
		
	8:
		// 지그 개방 (액츄에이터 기동)
		IF EISIndex = 0 THEN
			ActuIndex:=12;
			ActuMove:=TO_INT(EISmove_csv[EISIndex,3]);
			Open_Serial:=TRUE;
			EISRetrieve_Seq:=9;
		ELSIF EISIndex=1 THEN
			ActuIndex:=11;
			ActuMove:=TO_INT(EISmove_csv[EISIndex,3]);
			Open_Serial:=TRUE;
			EISRetrieve_Seq:=9;
		END_IF;
		
	9:
		// 액츄에이터 통신 종료 확인 및 3s 기다림
		IF NOT Serial_Busy THEN
			Delay_TON13.In := TRUE;
			Delay_TON13.PT := T#1s;
			Delay_TON13();
			
			IF Delay_TON13.Q THEN
				Delay_TON13.In := FALSE;
				Delay_TON13();
				EISRetrieve_Seq:= 10;
			END_IF;
		END_IF;
		
	10:
		// 액츄에이터 회수
		ActuIndex:=13;
		ActuMove:=0;
		Open_Serial:=TRUE;	
		EISRetrieve_Seq:=11;
		
	11:
		// 액츄에이터 통신 종료 확인 및 3s 기다림
		IF NOT Serial_Busy THEN
			Delay_TON13.In := TRUE;
			Delay_TON13.PT := T#1s;
			Delay_TON13();
			
			IF Delay_TON13.Q THEN
				Delay_TON13.In := FALSE;
				Delay_TON13();
				EISRetrieve_Seq:= 12;
			END_IF;
		END_IF;
	
	12:
		// 지그 폐쇄 (액츄에이터 기동)
		IF EISIndex = 0 THEN
			ActuIndex:=12;
		ELSIF EISIndex=1 THEN
			ActuIndex:=11;
		END_IF;
		ActuMove:=0;
		Open_Serial:=TRUE;
		EISRetrieve_Seq:=13;
		
	13:
		// 액츄에이터 통신 종료 확인 및 0.5s 기다림
		Finish5:=FALSE;
		
		IF NOT Serial_Busy THEN
			Delay_TON13.In := TRUE;
			Delay_TON13.PT := T#1s;
			Delay_TON13();
			
			IF Delay_TON13.Q THEN
				Delay_TON13.In := FALSE;
				Delay_TON13();
				EISRetrieve_Seq:= 14;
			END_IF;
		END_IF;
	
	14:
		// 왼쪽으로 이동
		IF EISIndex=0 THEN
			Motor5_Move:=-850;
			Motor5_Check:=TRUE;
			EISRetrieve_Seq:=15;
		ELSIF EISIndex=1 THEN
			Motor5_Move:=-1250;
			Motor5_Check:=TRUE;
			EISRetrieve_Seq:=15;
		END_IF;
		
	15:
		// 0.5s 대기
		Delay_TON13.In := TRUE;
		Delay_TON13.PT := T#0.5s;
		Delay_TON13();
		
		IF Delay_TON13.Q THEN
			Delay_TON13.In := FALSE;
			Delay_TON13();
			EISRetrieve_Seq:= 16;
		END_IF;
		
	16:
		// 원점 복귀
		IF Finish5 THEN
			Finish5:=FALSE;
			Finish7:=FALSE;
			Jig_Origin:=TRUE;
			EISRetrieve_Seq:=17;
		END_IF;
		
	17:
		IF Finish5 AND Finish7 THEN
			JOB_Done:=TRUE;
			EISRetrieve_Seq:=0;
		END_IF;

END_CASE;

(* Section Section4: ladder, written here as Structured Text *)

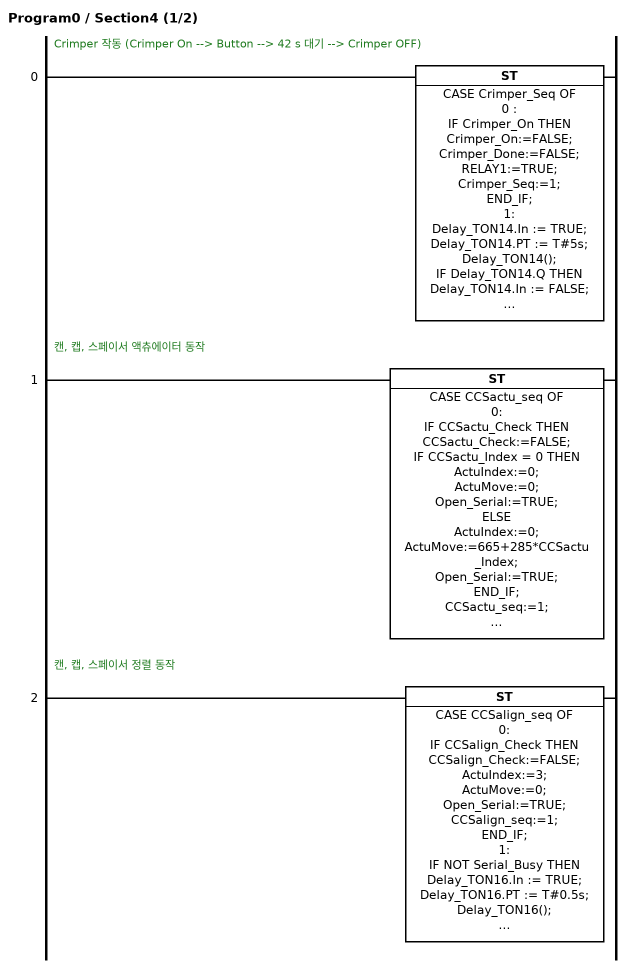
(* Rung 0: Crimper 작동 (Crimper On --> Button --> 42 s 대기 --> Crimper OFF) *)
CASE Crimper_Seq OF
    0 : 
		IF Crimper_On THEN
			Crimper_On:=FALSE;
			Crimper_Done:=FALSE;
			RELAY1:=TRUE;
			Crimper_Seq:=1;
		END_IF;
	
	1:
		Delay_TON14.In := TRUE;
		Delay_TON14.PT := T#5s;
		Delay_TON14();
			
		IF Delay_TON14.Q THEN
			Delay_TON14.In := FALSE;
			Delay_TON14();
			Crimper_Seq:= 2;
		END_IF;
	
	2:
		// 액츄에이터 기동 (버튼 누름)
		ActuIndex:=8;
		ActuMove:=1200;
		Open_Serial:=TRUE;
		Crimper_Seq:=3;
		
	3:
		// 액츄에이터 통신 종료 확인 및 1s 기다림
		IF NOT Serial_Busy THEN
			Delay_TON14.In := TRUE;
			Delay_TON14.PT := T#2s;
			Delay_TON14();
			
			IF Delay_TON14.Q THEN
				Delay_TON14.In := FALSE;
				Delay_TON14();
				Crimper_Seq:= 4;
			END_IF;
		END_IF;
		
	4:
		// 액츄에이터 기동 (버튼 누름)
		ActuIndex:=8;
		ActuMove:=0;
		Open_Serial:=TRUE;
		Crimper_Seq:=5;
		
	5:
		// 액츄에이터 통신 종료 확인 및 42s 기다림
		IF NOT Serial_Busy THEN
			Delay_TON14.In := TRUE;
			Delay_TON14.PT := T#42s;
			Delay_TON14();
			
			IF Delay_TON14.Q THEN
				Delay_TON14.In := FALSE;
				Delay_TON14();
				Crimper_Seq:= 6;
			END_IF;
		END_IF;
		
	6:
		RELAY1:=FALSE;
		Crimper_Done:=TRUE;
		Crimper_Seq:=0;
		
END_CASE;
(* Rung 1: 캔, 캡, 스페이서 액츄에이터 동작 *)
CASE CCSactu_seq OF
	0:
		IF CCSactu_Check THEN
			CCSactu_Check:=FALSE;
			IF CCSactu_Index = 0 THEN
				ActuIndex:=0;
				ActuMove:=0;
				Open_Serial:=TRUE;
			ELSE
				ActuIndex:=0;
				ActuMove:=665+285*CCSactu_Index;
				Open_Serial:=TRUE;
			END_IF;
			CCSactu_seq:=1;
		END_IF;
	
	1:
		// 액츄에이터 통신 종료 확인 및 1s 기다림
		IF NOT Serial_Busy THEN
			Delay_TON15.In := TRUE;
			Delay_TON15.PT := T#0.5s;
			Delay_TON15();
			
			IF Delay_TON15.Q THEN
				Delay_TON15.In := FALSE;
				Delay_TON15();
				CCSactu_seq:= 2;
			END_IF;
		END_IF;
	
	2:
		IF CCSactu_Index = 0 THEN
			ActuIndex:=1;
			ActuMove:=0;
			Open_Serial:=TRUE;
		ELSE
			ActuIndex:=1;
			ActuMove:=665+285*CCSactu_Index;
			Open_Serial:=TRUE;
		END_IF;
		CCSactu_seq:=3;
	
	3:
		// 액츄에이터 통신 종료 확인 및 1s 기다림
		IF NOT Serial_Busy THEN
			Delay_TON15.In := TRUE;
			Delay_TON15.PT := T#0.5s;
			Delay_TON15();
			
			IF Delay_TON15.Q THEN
				Delay_TON15.In := FALSE;
				Delay_TON15();
				CCSactu_seq:= 4;
			END_IF;
		END_IF;
	
	4:
		IF CCSactu_Index = 0 THEN
			ActuIndex:=2;
			ActuMove:=0;
			Open_Serial:=TRUE;
		ELSE
			ActuIndex:=2;
			ActuMove:=1975+135*CCSactu_Index;
			Open_Serial:=TRUE;
		END_IF;
		CCSactu_seq:=0;
			
END_CASE;
(* Rung 2: 캔, 캡, 스페이서 정렬 동작 *)
CASE CCSalign_seq OF
	0:
		IF CCSalign_Check THEN
			CCSalign_Check:=FALSE;
			ActuIndex:=3;
			ActuMove:=0;
			Open_Serial:=TRUE;
			CCSalign_seq:=1;
		END_IF;
		
	1:
		IF NOT Serial_Busy THEN
			Delay_TON16.In := TRUE;
			Delay_TON16.PT := T#0.5s;
			Delay_TON16();
			
			IF Delay_TON16.Q THEN
				Delay_TON16.In := FALSE;
				Delay_TON16();
				CCSalign_seq:= 2;
			END_IF;
		END_IF;
		
	2:
		ActuIndex:=3;
		ActuMove:=1150;
		Open_Serial:=TRUE;
		CCSalign_seq:=3;
		
	3:
		IF NOT Serial_Busy THEN
			Delay_TON16.In := TRUE;
			Delay_TON16.PT := T#0.5s;
			Delay_TON16();
			
			IF Delay_TON16.Q THEN
				Delay_TON16.In := FALSE;
				Delay_TON16();
				CCSalign_seq:= 4;
			END_IF;
		END_IF;
		
	4:
		ActuIndex:=3;
		ActuMove:=0;
		Open_Serial:=TRUE;
		CCSalign_seq:=5;
		
	5:
		IF NOT Serial_Busy THEN
			Delay_TON16.In := TRUE;
			Delay_TON16.PT := T#0.5s;
			Delay_TON16();
			
			IF Delay_TON16.Q THEN
				Delay_TON16.In := FALSE;
				Delay_TON16();
				CCSalign_seq:= 6;
			END_IF;
		END_IF;
		
	6:
		ActuIndex:=3;
		ActuMove:=1200;
		Open_Serial:=TRUE;
		CCSalign_seq:=0;
		
END_CASE;

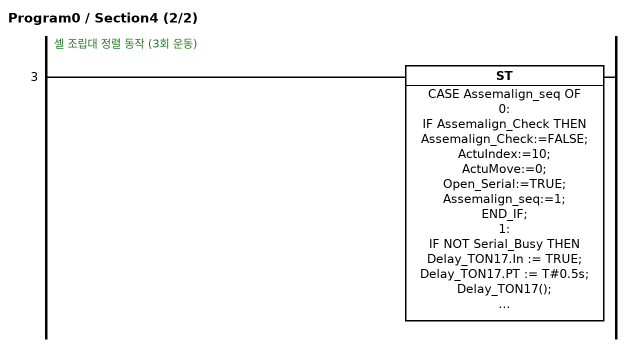
(* Rung 3: 셀 조립대 정렬 동작 (3회 운동) *)
CASE Assemalign_seq OF
	0:
		IF Assemalign_Check THEN
			Assemalign_Check:=FALSE;
			ActuIndex:=10;
			ActuMove:=0;
			Open_Serial:=TRUE;
			Assemalign_seq:=1;
		END_IF;
		
	1:
		IF NOT Serial_Busy THEN
			Delay_TON17.In := TRUE;
			Delay_TON17.PT := T#0.5s;
			Delay_TON17();
			
			IF Delay_TON17.Q THEN
				Delay_TON17.In := FALSE;
				Delay_TON17();
				Assemalign_seq:= 2;
			END_IF;
		END_IF;
		
	2:
		ActuIndex:=10;
		ActuMove:=500;
		Open_Serial:=TRUE;
		Assemalign_seq:=3;
		
	3:
		IF NOT Serial_Busy THEN
			Delay_TON17.In := TRUE;
			Delay_TON17.PT := T#0.5s;
			Delay_TON17();
			
			IF Delay_TON17.Q THEN
				Delay_TON17.In := FALSE;
				Delay_TON17();
				Assemalign_seq:= 4;
			END_IF;
		END_IF;
		
	4:
		ActuIndex:=10;
		ActuMove:=0;
		Open_Serial:=TRUE;
		Assemalign_seq:=5;
		
	5:
		IF NOT Serial_Busy THEN
			Delay_TON17.In := TRUE;
			Delay_TON17.PT := T#0.5s;
			Delay_TON17();
			
			IF Delay_TON17.Q THEN
				Delay_TON17.In := FALSE;
				Delay_TON17();
				Assemalign_seq:= 6;
			END_IF;
		END_IF;
		
	6:
		ActuIndex:=10;
		ActuMove:=500;
		Open_Serial:=TRUE;
		Assemalign_seq:=7;
		
	7:
		IF NOT Serial_Busy THEN
			Delay_TON17.In := TRUE;
			Delay_TON17.PT := T#0.5s;
			Delay_TON17();
			
			IF Delay_TON17.Q THEN
				Delay_TON17.In := FALSE;
				Delay_TON17();
				Assemalign_seq:= 8;
			END_IF;
		END_IF;
		
	8:
		ActuIndex:=10;
		ActuMove:=0;
		Open_Serial:=TRUE;
		Assemalign_seq:=0;
		
END_CASE;

(* Section Section5: ladder, written here as Structured Text *)

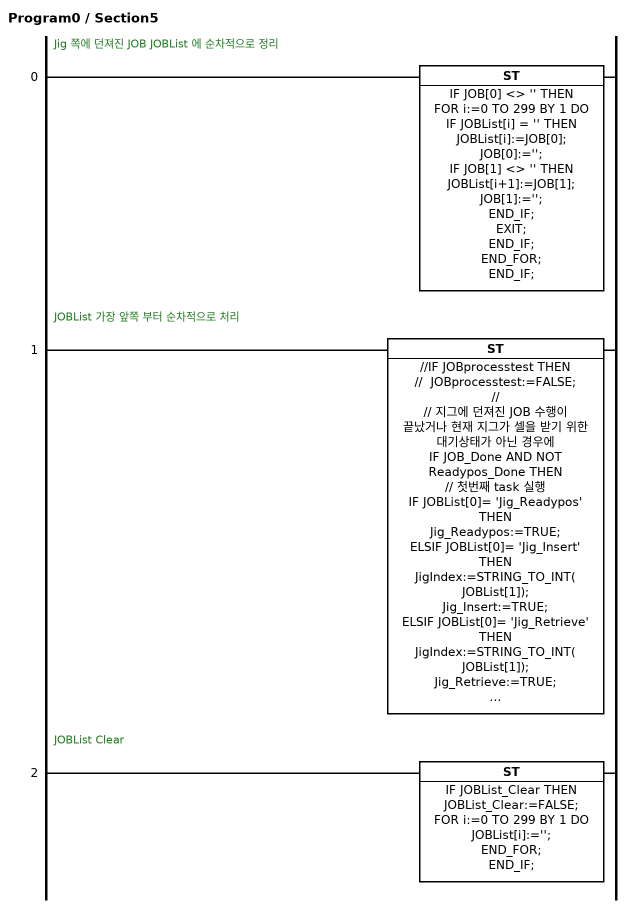
(* Rung 0: Jig 쪽에 던져진 JOB JOBList 에 순차적으로 정리 *)
IF JOB[0] <> '' THEN
		FOR i:=0 TO 299 BY 1 DO
			IF JOBList[i] = '' THEN
				JOBList[i]:=JOB[0];
				JOB[0]:='';
				IF JOB[1] <> '' THEN
					JOBList[i+1]:=JOB[1];
					JOB[1]:='';
				END_IF;
				EXIT;
			END_IF;
		END_FOR;
END_IF;
(* Rung 1: JOBList 가장 앞쪽 부터 순차적으로 처리 *)
//IF JOBprocesstest THEN
//	JOBprocesstest:=FALSE;
//
// 지그에 던져진 JOB 수행이 끝났거나 현재 지그가 셀을 받기 위한 대기상태가 아닌 경우에
IF JOB_Done AND NOT Readypos_Done THEN
	
	// 첫번째 task 실행 
	IF JOBList[0]= 'Jig_Readypos' THEN
		Jig_Readypos:=TRUE;
	ELSIF JOBList[0]= 'Jig_Insert' THEN
		JigIndex:=STRING_TO_INT(JOBList[1]);
		Jig_Insert:=TRUE;
	ELSIF JOBList[0]= 'Jig_Retrieve' THEN
		JigIndex:=STRING_TO_INT(JOBList[1]);
		Jig_Retrieve:=TRUE;
	ELSIF JOBList[0]= 'EIS_Insert' THEN
		EISIndex:=STRING_TO_INT(JOBList[1]);
		EIS_Insert:=TRUE;
	ELSIF JOBList[0]= 'EIS_Retrieve' THEN
		EISIndex:=STRING_TO_INT(JOBList[1]);
		EIS_Retrieve:=TRUE;
	END_IF;
	
	// 첫번째 task DataJig 에 반영 후 제거
	DataJig.Gantry[0]:=JOBList[0];
	DataJig.Gantry[1]:=JOBList[1];
	JOBList[0]:='';
	JOBList[1]:='';
	
	// 앞으로 한칸씩 당기기
	FOR i:=2 TO 299 BY 1 DO
		JOBList[i-2]:=JOBList[i];
	END_FOR;
	
END_IF;
(* Rung 2: JOBList Clear *)
IF JOBList_Clear THEN
	JOBList_Clear:=FALSE;
	FOR i:=0 TO 299 BY 1 DO
		JOBList[i]:=''; 
	END_FOR;
END_IF;
END_PROGRAM

FUNCTION_BLOCK STEPmotor
VAR
    PCount : INT := 0;
    PulseTON1 : TON;
    PulseTON2 : TON;
    o : BOOL;
END_VAR
VAR_INPUT
    Enable : BOOL;
    StepControl : sStepControl;
END_VAR
VAR_IN_OUT
    Direction : BOOL;
    Pulse : BOOL;
END_VAR
VAR_OUTPUT
    Done : BOOL;
    Moving : BOOL;
END_VAR
VAR_IN_OUT
    Finish : BOOL;
END_VAR
VAR_EXTERNAL
    Direction0 : BOOL;
    Pulse0 : BOOL;
    Pulse1 : BOOL;
    Pulse2 : BOOL;
    Direction2 : BOOL;
    Direction1 : BOOL;
    Direction3 : BOOL;
    Pulse3 : BOOL;
END_VAR
VAR
    _e1 : R_TRIG;
    _p2 : BOOL;
    _e3 : R_TRIG;
    _e4 : F_TRIG;
END_VAR
(* ladder, written here as Structured Text *)

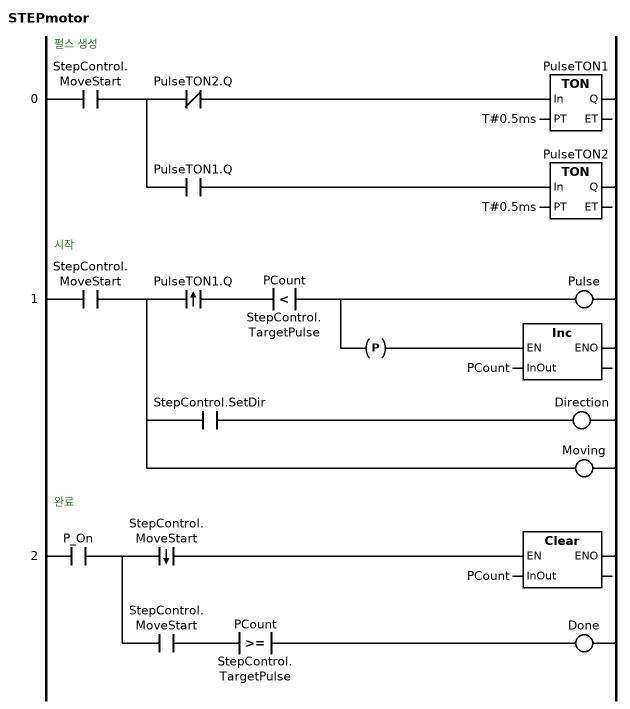
(* Rung 0: 펄스 생성 *)
PulseTON1(In := StepControl.MoveStart AND NOT PulseTON2.Q, PT := T#0.5ms);
PulseTON2(In := StepControl.MoveStart AND PulseTON1.Q, PT := T#0.5ms);
(* Rung 1: 시작 *)
_e1(CLK := PulseTON1.Q);
_p2 := StepControl.MoveStart AND _e1.Q AND (PCount < StepControl.TargetPulse);
Pulse := _p2;
_e3(CLK := _p2);
IF _e3.Q THEN Inc(InOut := PCount); END_IF;
Direction := StepControl.MoveStart AND StepControl.SetDir;
Moving := StepControl.MoveStart;
(* Rung 2: 완료 *)
_e4(CLK := StepControl.MoveStart);
IF P_On AND _e4.Q THEN Clear(InOut := PCount); END_IF;
Done := P_On AND StepControl.MoveStart AND (PCount >= StepControl.TargetPulse);
END_FUNCTION_BLOCK